LIN {X 0,Y 316.148,Z 1080.606,A -85,B 0,C 180,E1 25715.482,E2 25715.482} C_VEL
LIN {X 0,Y 359.613,Z 1022.484,A -85,B 0,C 180,E1 25721.601,E2 25721.601} C_VEL
LIN {X 0,Y 369.692,Z 1005.378,A -85,B 0,C 180,E1 25723.065,E2 25723.065} C_VEL
LIN {X 0,Y 370.148,Z 988.443,A -85,B 0,C 180,E1 25731.773,E2 25731.773} C_VEL
LIN {X 0,Y 370.715,Z 983.832,A -85,B 0,C 180,E1 25738.851,E2 25738.851} C_VEL
LIN {X 0,Y 369.808,Z 994.61,A -85,B 0,C 180,E1 25748.283,E2 25748.283} C_VEL
LIN {X 0,Y 368.373,Z 1009.498,A -85,B 0,C 180,E1 25754.057,E2 25754.057} C_VEL
LIN {X 0,Y 326.146,Z 1071.026,A -85,B 0,C 180,E1 25759.675,E2 25759.675} C_VEL
LIN {X 0,Y 280.052,Z 1123.121,A -85,B 0,C 180,E1 25768.626,E2 25768.626} C_VEL
LIN {X 0,Y 237.395,Z 1163.97,A -85,B 0,C 180,E1 25782.718,E2 25782.718} C_VEL
LIN {X 0,Y 210.63,Z 1190.183,A -85,B 0,C 180,E1 25802.091,E2 25802.091} C_VEL
LIN {X 0,Y 203.395,Z 1200.362,A -85,B 0,C 180,E1 25819.253,E2 25819.253} C_VEL
LIN {X 0,Y 203.105,Z 1202.001,A -85,B 0,C 180,E1 25832.135,E2 25832.135} C_VEL
LIN {X 0,Y 205.625,Z 1196.351,A -85,B 0,C 180,E1 25849.379,E2 25849.379} C_VEL
LIN {X 0,Y 224.205,Z 1176.349,A -85,B 0,C 180,E1 25869.979,E2 25869.979} C_VEL
LIN {X 0,Y 261.978,Z 1141.015,A -85,B 0,C 180,E1 25886.466,E2 25886.466} C_VEL
LIN {X 0,Y 308.24,Z 1092.884,A -85,B 0,C 180,E1 25897.284,E2 25897.284} C_VEL
LIN {X 0,Y 353.537,Z 1033.592,A -85,B 0,C 180,E1 25904.178,E2 25904.178} C_VEL
LIN {X 0,Y 369.486,Z 1007.292,A -85,B 0,C 180,E1 25906.321,E2 25906.321} C_VEL
LIN {X 0,Y 370.03,Z 990.826,A -85,B 0,C 180,E1 25914.09,E2 25914.09} C_VEL
LIN {X 0,Y 371.036,Z 983.808,A -85,B 0,C 180,E1 25921.148,E2 25921.148} C_VEL
LIN {X 0,Y 370.096,Z 993.398,A -85,B 0,C 180,E1 25931.209,E2 25931.209} C_VEL
LIN {X 0,Y 368.996,Z 1007.618,A -85,B 0,C 180,E1 25937.205,E2 25937.205} C_VEL
LIN {X 0,Y 326.774,Z 1068.114,A -85,B 0,C 180,E1 25942.732,E2 25942.732} C_VEL
LIN {X 0,Y 293.393,Z 1105.685,A -85,B 0,C 180,E1 25948.682,E2 25948.682} C_VEL
LIN {X 0,Y 268.809,Z 1125.767,A -85,B 0,C 180,E1 25951.921,E2 25951.921} C_VEL
LIN {X 0,Y 226.225,Z 1161.867,A -85,B 0,C 180,E1 25966.765,E2 25966.765} C_VEL
LIN {X 0,Y 202.01,Z 1181.995,A -85,B 0,C 180,E1 25985.618,E2 25985.618} C_VEL
LIN {X 0,Y 195.444,Z 1189.255,A -85,B 0,C 180,E1 26003.321,E2 26003.321} C_VEL
LIN {X 0,Y 195.404,Z 1189.222,A -85,B 0,C 180,E1 26016.69,E2 26016.69} C_VEL
LIN {X 0,Y 204.145,Z 1180,A -85,B 0,C 180,E1 26037.107,E2 26037.107} C_VEL
LIN {X 0,Y 234.232,Z 1155.422,A -85,B 0,C 180,E1 26056.755,E2 26056.755} C_VEL
LIN {X 0,Y 277.988,Z 1117.112,A -85,B 0,C 180,E1 26070.177,E2 26070.177} C_VEL
LIN {X 0,Y 325.42,Z 1066.08,A -85,B 0,C 180,E1 26078.761,E2 26078.761} C_VEL
LIN {X 0,Y 364.954,Z 1010.019,A -85,B 0,C 180,E1 26083.947,E2 26083.947} C_VEL
LIN {X 0,Y 365.855,Z 995.479,A -85,B 0,C 180,E1 26091.676,E2 26091.676} C_VEL
LIN {X 0,Y 366.492,Z 990.687,A -85,B 0,C 180,E1 26098.838,E2 26098.838} C_VEL
LIN {X 0,Y 365.305,Z 1001.773,A -85,B 0,C 180,E1 26108.386,E2 26108.386} C_VEL
LIN {X 0,Y 363.604,Z 1013.922,A -85,B 0,C 180,E1 26113.125,E2 26113.125} C_VEL
LIN {X 0,Y 318.765,Z 1076.531,A -85,B 0,C 180,E1 26118.987,E2 26118.987} C_VEL
LIN {X 0,Y 271.684,Z 1127.247,A -85,B 0,C 180,E1 26128.161,E2 26128.161} C_VEL
LIN {X 0,Y 227.974,Z 1166.993,A -85,B 0,C 180,E1 26142.962,E2 26142.962} C_VEL
LIN {X 0,Y 201.693,Z 1191.616,A -85,B 0,C 180,E1 26163.179,E2 26163.179} C_VEL
LIN {X 0,Y 195.081,Z 1201.22,A -85,B 0,C 180,E1 26183.299,E2 26183.299} C_VEL
LIN {X 0,Y 195.077,Z 1201.233,A -85,B 0,C 180,E1 26196.692,E2 26196.692} C_VEL
LIN {X 0,Y 200.185,Z 1193.301,A -85,B 0,C 180,E1 26214.619,E2 26214.619} C_VEL
LIN {X 0,Y 224.297,Z 1170.256,A -85,B 0,C 180,E1 26235.223,E2 26235.223} C_VEL
LIN {X 0,Y 265.902,Z 1132.749,A -85,B 0,C 180,E1 26250.423,E2 26250.423} C_VEL
LIN {X 0,Y 314.147,Z 1082.127,A -85,B 0,C 180,E1 26260.27,E2 26260.27} C_VEL
LIN {X 0,Y 359.015,Z 1021.48,A -85,B 0,C 180,E1 26266.376,E2 26266.376} C_VEL
LIN {X 0,Y 364.771,Z 1011.464,A -85,B 0,C 180,E1 26267.357,E2 26267.357} C_VEL
LIN {X 0,Y 365.816,Z 996.158,A -85,B 0,C 180,E1 26275.216,E2 26275.216} C_VEL
LIN {X 0,Y 366.821,Z 990.653,A -85,B 0,C 180,E1 26281.161,E2 26281.161} C_VEL
LIN {X 0,Y 365.711,Z 999.528,A -85,B 0,C 180,E1 26290.739,E2 26290.739} C_VEL
LIN {X 0,Y 364.587,Z 1011.509,A -85,B 0,C 180,E1 26296.224,E2 26296.224} C_VEL
LIN {X 0,Y 320.68,Z 1072.197,A -85,B 0,C 180,E1 26301.87,E2 26301.87} C_VEL
LIN {X 0,Y 273.521,Z 1121.485,A -85,B 0,C 180,E1 26310.759,E2 26310.759} C_VEL
LIN {X 0,Y 268.809,Z 1125.767,A -85,B 0,C 180,E1 26311.921,E2 26311.921} C_VEL
LIN {X 0,Y 244.101,Z 1143.39,A -85,B 0,C 180,E1 26316.075,E2 26316.075} C_VEL
LIN {X 0,Y 205.94,Z 1173.133,A -85,B 0,C 180,E1 26333.787,E2 26333.787} C_VEL
LIN {X 0,Y 189.446,Z 1186.942,A -85,B 0,C 180,E1 26353.734,E2 26353.734} C_VEL
LIN {X 0,Y 187.43,Z 1189.94,A -85,B 0,C 180,E1 26372.323,E2 26372.323} C_VEL
LIN {X 0,Y 192.941,Z 1183.622,A -85,B 0,C 180,E1 26393.146,E2 26393.146} C_VEL
LIN {X 0,Y 218.988,Z 1163.089,A -85,B 0,C 180,E1 26413.976,E2 26413.976} C_VEL
LIN {X 0,Y 262.449,Z 1127.725,A -85,B 0,C 180,E1 26429.025,E2 26429.025} C_VEL
LIN {X 0,Y 311.303,Z 1079.422,A -85,B 0,C 180,E1 26438.481,E2 26438.481} C_VEL
LIN {X 0,Y 356.624,Z 1020.527,A -85,B 0,C 180,E1 26444.269,E2 26444.269} C_VEL
LIN {X 0,Y 360.249,Z 1014.774,A -85,B 0,C 180,E1 26444.806,E2 26444.806} C_VEL
LIN {X 0,Y 361.457,Z 1001.135,A -85,B 0,C 180,E1 26452.788,E2 26452.788} C_VEL
LIN {X 0,Y 362.265,Z 997.544,A -85,B 0,C 180,E1 26458.824,E2 26458.824} C_VEL
LIN {X 0,Y 360.713,Z 1007.612,A -85,B 0,C 180,E1 26467.885,E2 26467.885} C_VEL
LIN {X 0,Y 358.795,Z 1018.34,A -85,B 0,C 180,E1 26472.177,E2 26472.177} C_VEL
LIN {X 0,Y 312.986,Z 1079.796,A -85,B 0,C 180,E1 26478.022,E2 26478.022} C_VEL
LIN {X 0,Y 264.611,Z 1129.862,A -85,B 0,C 180,E1 26487.33,E2 26487.33} C_VEL
LIN {X 0,Y 220.325,Z 1168.374,A -85,B 0,C 180,E1 26502.322,E2 26502.322} C_VEL
LIN {X 0,Y 194.323,Z 1191.359,A -85,B 0,C 180,E1 26522.075,E2 26522.075} C_VEL
LIN {X 0,Y 187.07,Z 1200.971,A -85,B 0,C 180,E1 26543.011,E2 26543.011} C_VEL
LIN {X 0,Y 187.066,Z 1200.984,A -85,B 0,C 180,E1 26556.98,E2 26556.98} C_VEL
LIN {X 0,Y 192.676,Z 1193.044,A -85,B 0,C 180,E1 26575.646,E2 26575.646} C_VEL
LIN {X 0,Y 218.416,Z 1169.988,A -85,B 0,C 180,E1 26596.8,E2 26596.8} C_VEL
LIN {X 0,Y 261.83,Z 1132.468,A -85,B 0,C 180,E1 26612.033,E2 26612.033} C_VEL
LIN {X 0,Y 311.426,Z 1081.82,A -85,B 0,C 180,E1 26621.717,E2 26621.717} C_VEL
LIN {X 0,Y 357.409,Z 1020.732,A -85,B 0,C 180,E1 26627.691,E2 26627.691} C_VEL
LIN {X 0,Y 360.11,Z 1015.85,A -85,B 0,C 180,E1 26628.363,E2 26628.363} C_VEL
LIN {X 0,Y 361.546,Z 1001.58,A -85,B 0,C 180,E1 26636.365,E2 26636.365} C_VEL
LIN {X 0,Y 362.6,Z 997.505,A -85,B 0,C 180,E1 26641.175,E2 26641.175} C_VEL
LIN {X 0,Y 361.062,Z 1006.48,A -85,B 0,C 180,E1 26650.879,E2 26650.879} C_VEL
LIN {X 0,Y 359.569,Z 1016.385,A -85,B 0,C 180,E1 26655.305,E2 26655.305} C_VEL
LIN {X 0,Y 314.729,Z 1075.84,A -85,B 0,C 180,E1 26660.939,E2 26660.939} C_VEL
LIN {X 0,Y 266.707,Z 1124.112,A -85,B 0,C 180,E1 26669.88,E2 26669.88} C_VEL
LIN {X 0,Y 244.101,Z 1143.39,A -85,B 0,C 180,E1 26676.075,E2 26676.075} C_VEL
LIN {X 0,Y 219.813,Z 1158.391,A -85,B 0,C 180,E1 26681.306,E2 26681.306} C_VEL
LIN {X 0,Y 188.769,Z 1181.284,A -85,B 0,C 180,E1 26701.682,E2 26701.682} C_VEL
LIN {X 0,Y 179.487,Z 1189.751,A -85,B 0,C 180,E1 26722.724,E2 26722.724} C_VEL
LIN {X 0,Y 179.428,Z 1189.721,A -85,B 0,C 180,E1 26737.288,E2 26737.288} C_VEL
LIN {X 0,Y 188.648,Z 1181.254,A -85,B 0,C 180,E1 26758.235,E2 26758.235} C_VEL
LIN {X 0,Y 219.961,Z 1158.336,A -85,B 0,C 180,E1 26778.52,E2 26778.52} C_VEL
LIN {X 0,Y 265.657,Z 1121.739,A -85,B 0,C 180,E1 26792.237,E2 26792.237} C_VEL
LIN {X 0,Y 315.107,Z 1072.386,A -85,B 0,C 180,E1 26800.828,E2 26800.828} C_VEL
LIN {X 0,Y 355.471,Z 1019.161,A -85,B 0,C 180,E1 26805.802,E2 26805.802} C_VEL
LIN {X 0,Y 356.974,Z 1006.833,A -85,B 0,C 180,E1 26813.923,E2 26813.923} C_VEL
LIN {X 0,Y 357.809,Z 1004.236,A -85,B 0,C 180,E1 26818.81,E2 26818.81} C_VEL
LIN {X 0,Y 355.979,Z 1014.642,A -85,B 0,C 180,E1 26827.99,E2 26827.99} C_VEL
LIN {X 0,Y 353.349,Z 1023.665,A -85,B 0,C 180,E1 26831.284,E2 26831.284} C_VEL
LIN {X 0,Y 306.092,Z 1084.408,A -85,B 0,C 180,E1 26837.196,E2 26837.196} C_VEL
LIN {X 0,Y 255.588,Z 1134.273,A -85,B 0,C 180,E1 26846.934,E2 26846.934} C_VEL
LIN {X 0,Y 210.554,Z 1171.596,A -85,B 0,C 180,E1 26862.763,E2 26862.763} C_VEL
LIN {X 0,Y 184.361,Z 1193.782,A -85,B 0,C 180,E1 26884.749,E2 26884.749} C_VEL
LIN {X 0,Y 179.061,Z 1200.721,A -85,B 0,C 180,E1 26902.697,E2 26902.697} C_VEL
LIN {X 0,Y 179.057,Z 1200.734,A -85,B 0,C 180,E1 26917.294,E2 26917.294} C_VEL
LIN {X 0,Y 185.211,Z 1192.786,A -85,B 0,C 180,E1 26936.76,E2 26936.76} C_VEL
LIN {X 0,Y 211.478,Z 1170.765,A -85,B 0,C 180,E1 26957.828,E2 26957.828} C_VEL
LIN {X 0,Y 256.495,Z 1133.534,A -85,B 0,C 180,E1 26973.322,E2 26973.322} C_VEL
LIN {X 0,Y 307.722,Z 1082.846,A -85,B 0,C 180,E1 26983.012,E2 26983.012} C_VEL
LIN {X 0,Y 354.488,Z 1022.232,A -85,B 0,C 180,E1 26988.865,E2 26988.865} C_VEL
LIN {X 0,Y 356.76,Z 1009.616,A -85,B 0,C 180,E1 26995.293,E2 26995.293} C_VEL
LIN {X 0,Y 358.136,Z 1004.212,A -85,B 0,C 180,E1 27001.189,E2 27001.189} C_VEL
LIN {X 0,Y 356.382,Z 1013.484,A -85,B 0,C 180,E1 27011.024,E2 27011.024} C_VEL
LIN {X 0,Y 354.227,Z 1021.652,A -85,B 0,C 180,E1 27014.403,E2 27014.403} C_VEL
LIN {X 0,Y 307.535,Z 1080.944,A -85,B 0,C 180,E1 27020.17,E2 27020.17} C_VEL
LIN {X 0,Y 258.599,Z 1127.919,A -85,B 0,C 180,E1 27029.278,E2 27029.278} C_VEL
LIN {X 0,Y 219.813,Z 1158.391,A -85,B 0,C 180,E1 27041.306,E2 27041.306} C_VEL
LIN {X 0,Y 197.353,Z 1170.633,A -85,B 0,C 180,E1 27048.102,E2 27048.102} C_VEL
LIN {X 0,Y 175.069,Z 1186.508,A -85,B 0,C 180,E1 27069.732,E2 27069.732} C_VEL
LIN {X 0,Y 171.299,Z 1190.45,A -85,B 0,C 180,E1 27087.468,E2 27087.468} C_VEL
LIN {X 0,Y 174.006,Z 1187.386,A -85,B 0,C 180,E1 27107.766,E2 27107.766} C_VEL
LIN {X 0,Y 195.922,Z 1171.396,A -85,B 0,C 180,E1 27131.148,E2 27131.148} C_VEL
LIN {X 0,Y 237.45,Z 1141.724,A -85,B 0,C 180,E1 27147.944,E2 27147.944} C_VEL
LIN {X 0,Y 288.79,Z 1097.502,A -85,B 0,C 180,E1 27158.773,E2 27158.773} C_VEL
LIN {X 0,Y 338.132,Z 1041.454,A -85,B 0,C 180,E1 27165.325,E2 27165.325} C_VEL
LIN {X 0,Y 350.672,Z 1023.964,A -85,B 0,C 180,E1 27166.674,E2 27166.674} C_VEL
LIN {X 0,Y 352.423,Z 1013.558,A -85,B 0,C 180,E1 27173.844,E2 27173.844} C_VEL
LIN {X 0,Y 353.285,Z 1010.885,A -85,B 0,C 180,E1 27178.794,E2 27178.794} C_VEL
LIN {X 0,Y 350.984,Z 1021.49,A -85,B 0,C 180,E1 27188.105,E2 27188.105} C_VEL
LIN {X 0,Y 348.689,Z 1027.918,A -85,B 0,C 180,E1 27190.271,E2 27190.271} C_VEL
LIN {X 0,Y 300.52,Z 1087.644,A -85,B 0,C 180,E1 27196.159,E2 27196.159} C_VEL
LIN {X 0,Y 248.199,Z 1137.19,A -85,B 0,C 180,E1 27206.136,E2 27206.136} C_VEL
LIN {X 0,Y 203.005,Z 1172.745,A -85,B 0,C 180,E1 27222.015,E2 27222.015} C_VEL
LIN {X 0,Y 176.089,Z 1194.236,A -85,B 0,C 180,E1 27244.949,E2 27244.949} C_VEL
LIN {X 0,Y 171.066,Z 1200.471,A -85,B 0,C 180,E1 27262.353,E2 27262.353} C_VEL
LIN {X 0,Y 171.062,Z 1200.485,A -85,B 0,C 180,E1 27277.637,E2 27277.637} C_VEL
LIN {X 0,Y 177.851,Z 1192.53,A -85,B 0,C 180,E1 27297.962,E2 27297.962} C_VEL
LIN {X 0,Y 207.26,Z 1169.459,A -85,B 0,C 180,E1 27320.193,E2 27320.193} C_VEL
LIN {X 0,Y 255.166,Z 1131.238,A -85,B 0,C 180,E1 27335.556,E2 27335.556} C_VEL
LIN {X 0,Y 306.592,Z 1081.211,A -85,B 0,C 180,E1 27344.685,E2 27344.685} C_VEL
LIN {X 0,Y 350.515,Z 1025.296,A -85,B 0,C 180,E1 27350.067,E2 27350.067} C_VEL
LIN {X 0,Y 352.797,Z 1012.784,A -85,B 0,C 180,E1 27358.742,E2 27358.742} C_VEL
LIN {X 0,Y 352.914,Z 1012.124,A -85,B 0,C 180,E1 27363.674,E2 27363.674} C_VEL
LIN {X 0,Y 350.965,Z 1022.787,A -85,B 0,C 180,E1 27372.502,E2 27372.502} C_VEL
LIN {X 0,Y 349.511,Z 1026.126,A -85,B 0,C 180,E1 27373.417,E2 27373.417} C_VEL
LIN {X 0,Y 301.887,Z 1084.419,A -85,B 0,C 180,E1 27379.146,E2 27379.146} C_VEL
LIN {X 0,Y 250.529,Z 1131.65,A -85,B 0,C 180,E1 27388.639,E2 27388.639} C_VEL
LIN {X 0,Y 205.093,Z 1165.26,A -85,B 0,C 180,E1 27403.874,E2 27403.874} C_VEL
LIN {X 0,Y 197.353,Z 1170.633,A -85,B 0,C 180,E1 27408.102,E2 27408.102} C_VEL
LIN {X 0,Y 177.075,Z 1180.099,A -85,B 0,C 180,E1 27416.564,E2 27416.564} C_VEL
LIN {X 0,Y 164.44,Z 1189.285,A -85,B 0,C 180,E1 27436.676,E2 27436.676} C_VEL
LIN {X 0,Y 163.401,Z 1190.683,A -85,B 0,C 180,E1 27452.665,E2 27452.665} C_VEL
LIN {X 0,Y 170.599,Z 1184.429,A -85,B 0,C 180,E1 27476.273,E2 27476.273} C_VEL
LIN {X 0,Y 201.697,Z 1164.027,A -85,B 0,C 180,E1 27498.76,E2 27498.76} C_VEL
LIN {X 0,Y 249.635,Z 1129.369,A -85,B 0,C 180,E1 27513.651,E2 27513.651} C_VEL
LIN {X 0,Y 301.498,Z 1082.119,A -85,B 0,C 180,E1 27522.562,E2 27522.562} C_VEL
LIN {X 0,Y 346.074,Z 1027.998,A -85,B 0,C 180,E1 27527.996,E2 27527.996} C_VEL
LIN {X 0,Y 348.156,Z 1018.32,A -85,B 0,C 180,E1 27536.276,E2 27536.276} C_VEL
LIN {X 0,Y 347.866,Z 1019.205,A -85,B 0,C 180,E1 27541.276,E2 27541.276} C_VEL
LIN {X 0,Y 345.552,Z 1030.072,A -85,B 0,C 180,E1 27549.071,E2 27549.071} C_VEL
LIN {X 0,Y 295.713,Z 1090.045,A -85,B 0,C 180,E1 27554.976,E2 27554.976} C_VEL
LIN {X 0,Y 242.416,Z 1138.628,A -85,B 0,C 180,E1 27564.885,E2 27564.885} C_VEL
LIN {X 0,Y 194.887,Z 1174.275,A -85,B 0,C 180,E1 27581.513,E2 27581.513} C_VEL
LIN {X 0,Y 167.396,Z 1195.046,A -85,B 0,C 180,E1 27605.935,E2 27605.935} C_VEL
LIN {X 0,Y 163.212,Z 1200.763,A -85,B 0,C 180,E1 27627.332,E2 27627.332} C_VEL
LIN {X 0,Y 163.694,Z 1199.123,A -85,B 0,C 180,E1 27643.386,E2 27643.386} C_VEL
LIN {X 0,Y 178.726,Z 1185.905,A -85,B 0,C 180,E1 27667.958,E2 27667.958} C_VEL
LIN {X 0,Y 217.781,Z 1157.795,A -85,B 0,C 180,E1 27688.054,E2 27688.054} C_VEL
LIN {X 0,Y 269.121,Z 1115.976,A -85,B 0,C 180,E1 27700.702,E2 27700.702} C_VEL
LIN {X 0,Y 321.265,Z 1061.956,A -85,B 0,C 180,E1 27708.285,E2 27708.285} C_VEL
LIN {X 0,Y 345.857,Z 1029.699,A -85,B 0,C 180,E1 27711.138,E2 27711.138} C_VEL
LIN {X 0,Y 348.062,Z 1019.342,A -85,B 0,C 180,E1 27718.725,E2 27718.725} C_VEL
LIN {X 0,Y 348.201,Z 1018.692,A -85,B 0,C 180,E1 27723.723,E2 27723.723} C_VEL
LIN {X 0,Y 345.992,Z 1028.957,A -85,B 0,C 180,E1 27732.259,E2 27732.259} C_VEL
LIN {X 0,Y 296.664,Z 1087.399,A -85,B 0,C 180,E1 27738.035,E2 27738.035} C_VEL
LIN {X 0,Y 245.226,Z 1133.012,A -85,B 0,C 180,E1 27747.293,E2 27747.293} C_VEL
LIN {X 0,Y 197.439,Z 1166.813,A -85,B 0,C 180,E1 27763.146,E2 27763.146} C_VEL
LIN {X 0,Y 177.075,Z 1180.099,A -85,B 0,C 180,E1 27776.564,E2 27776.564} C_VEL
LIN {X 0,Y 160.31,Z 1186.702,A -85,B 0,C 180,E1 27786.989,E2 27786.989} C_VEL
LIN {X 0,Y 155.28,Z 1190.945,A -85,B 0,C 180,E1 27807.207,E2 27807.207} C_VEL
LIN {X 0,Y 158.613,Z 1187.888,A -85,B 0,C 180,E1 27829.556,E2 27829.556} C_VEL
LIN {X 0,Y 183.833,Z 1171.909,A -85,B 0,C 180,E1 27854.53,E2 27854.53} C_VEL
LIN {X 0,Y 228.902,Z 1142.399,A -85,B 0,C 180,E1 27871.39,E2 27871.39} C_VEL
LIN {X 0,Y 283.283,Z 1098.089,A -85,B 0,C 180,E1 27881.855,E2 27881.855} C_VEL
LIN {X 0,Y 334.214,Z 1042.379,A -85,B 0,C 180,E1 27887.997,E2 27887.997} C_VEL
LIN {X 0,Y 341.349,Z 1032.559,A -85,B 0,C 180,E1 27889.062,E2 27889.062} C_VEL
LIN {X 0,Y 343.423,Z 1024.484,A -85,B 0,C 180,E1 27897.097,E2 27897.097} C_VEL
LIN {X 0,Y 342.232,Z 1028.788,A -85,B 0,C 180,E1 27904.384,E2 27904.384} C_VEL
LIN {X 0,Y 340.123,Z 1035.463,A -85,B 0,C 180,E1 27908.143,E2 27908.143} C_VEL
LIN {X 0,Y 289.167,Z 1094.136,A -85,B 0,C 180,E1 27914.007,E2 27914.007} C_VEL
LIN {X 0,Y 234.775,Z 1141.61,A -85,B 0,C 180,E1 27924.061,E2 27924.061} C_VEL
LIN {X 0,Y 186.401,Z 1176.078,A -85,B 0,C 180,E1 27941.181,E2 27941.181} C_VEL
LIN {X 0,Y 159.909,Z 1194.791,A -85,B 0,C 180,E1 27964.732,E2 27964.732} C_VEL
LIN {X 0,Y 155.193,Z 1200.515,A -85,B 0,C 180,E1 27987.194,E2 27987.194} C_VEL
LIN {X 0,Y 155.786,Z 1198.872,A -85,B 0,C 180,E1 28004.079,E2 28004.079} C_VEL
LIN {X 0,Y 172.246,Z 1185.648,A -85,B 0,C 180,E1 28029.66,E2 28029.66} C_VEL
LIN {X 0,Y 215.14,Z 1156.359,A -85,B 0,C 180,E1 28050.512,E2 28050.512} C_VEL
LIN {X 0,Y 268.052,Z 1114.339,A -85,B 0,C 180,E1 28062.679,E2 28062.679} C_VEL
LIN {X 0,Y 320.643,Z 1060.484,A -85,B 0,C 180,E1 28069.851,E2 28069.851} C_VEL
LIN {X 0,Y 341.192,Z 1034.02,A -85,B 0,C 180,E1 28072.244,E2 28072.244} C_VEL
LIN {X 0,Y 344.158,Z 1023.885,A -85,B 0,C 180,E1 28081.238,E2 28081.238} C_VEL
LIN {X 0,Y 341.599,Z 1032.097,A -85,B 0,C 180,E1 28090.399,E2 28090.399} C_VEL
LIN {X 0,Y 338.689,Z 1036.85,A -85,B 0,C 180,E1 28091.51,E2 28091.51} C_VEL
LIN {X 0,Y 287.992,Z 1093.71,A -85,B 0,C 180,E1 28097.374,E2 28097.374} C_VEL
LIN {X 0,Y 234.647,Z 1138.428,A -85,B 0,C 180,E1 28107.175,E2 28107.175} C_VEL
LIN {X 0,Y 188.083,Z 1169.48,A -85,B 0,C 180,E1 28123.244,E2 28123.244} C_VEL
LIN {X 0,Y 160.31,Z 1186.702,A -85,B 0,C 180,E1 28146.989,E2 28146.989} C_VEL
LIN {X 0,Y 147.799,Z 1190.449,A -85,B 0,C 180,E1 28159.315,E2 28159.315} C_VEL
LIN {X 0,Y 147.555,Z 1190.716,A -85,B 0,C 180,E1 28178.874,E2 28178.874} C_VEL
LIN {X 0,Y 161.187,Z 1181.92,A -85,B 0,C 180,E1 28204.374,E2 28204.374} C_VEL
LIN {X 0,Y 201.291,Z 1158.378,A -85,B 0,C 180,E1 28226.229,E2 28226.229} C_VEL
LIN {X 0,Y 253.585,Z 1121.644,A -85,B 0,C 180,E1 28239.144,E2 28239.144} C_VEL
LIN {X 0,Y 307.659,Z 1071.746,A -85,B 0,C 180,E1 28246.807,E2 28246.807} C_VEL
LIN {X 0,Y 336.43,Z 1037.605,A -85,B 0,C 180,E1 28249.881,E2 28249.881} C_VEL
LIN {X 0,Y 339.02,Z 1030.333,A -85,B 0,C 180,E1 28258.744,E2 28258.744} C_VEL
LIN {X 0,Y 336.112,Z 1038.748,A -85,B 0,C 180,E1 28266.849,E2 28266.849} C_VEL
LIN {X 0,Y 283.878,Z 1097.101,A -85,B 0,C 180,E1 28272.841,E2 28272.841} C_VEL
LIN {X 0,Y 228.398,Z 1143.654,A -85,B 0,C 180,E1 28282.878,E2 28282.878} C_VEL
LIN {X 0,Y 179.728,Z 1176.629,A -85,B 0,C 180,E1 28299.808,E2 28299.808} C_VEL
LIN {X 0,Y 150.937,Z 1195.819,A -85,B 0,C 180,E1 28326.307,E2 28326.307} C_VEL
LIN {X 0,Y 147.162,Z 1200.267,A -85,B 0,C 180,E1 28347.041,E2 28347.041} C_VEL
LIN {X 0,Y 147.911,Z 1198.621,A -85,B 0,C 180,E1 28364.846,E2 28364.846} C_VEL
LIN {X 0,Y 165.904,Z 1185.39,A -85,B 0,C 180,E1 28391.5,E2 28391.5} C_VEL
LIN {X 0,Y 210.263,Z 1156.652,A -85,B 0,C 180,E1 28412.254,E2 28412.254} C_VEL
LIN {X 0,Y 265.007,Z 1114.613,A -85,B 0,C 180,E1 28424.301,E2 28424.301} C_VEL
LIN {X 0,Y 318.771,Z 1060.775,A -85,B 0,C 180,E1 28431.267,E2 28431.267} C_VEL
LIN {X 0,Y 336.315,Z 1038.815,A -85,B 0,C 180,E1 28433.17,E2 28433.17} C_VEL
LIN {X 0,Y 339.336,Z 1030.325,A -85,B 0,C 180,E1 28441.255,E2 28441.255} C_VEL
LIN {X 0,Y 336.497,Z 1037.893,A -85,B 0,C 180,E1 28450.066,E2 28450.066} C_VEL
LIN {X 0,Y 285.659,Z 1093.995,A -85,B 0,C 180,E1 28455.81,E2 28455.81} C_VEL
LIN {X 0,Y 231.888,Z 1138.032,A -85,B 0,C 180,E1 28465.137,E2 28465.137} C_VEL
LIN {X 0,Y 182.519,Z 1169.738,A -85,B 0,C 180,E1 28481.354,E2 28481.354} C_VEL
LIN {X 0,Y 152.408,Z 1187.262,A -85,B 0,C 180,E1 28506.552,E2 28506.552} C_VEL
LIN {X 0,Y 147.799,Z 1190.449,A -85,B 0,C 180,E1 28519.315,E2 28519.315} C_VEL
LIN {X 0,Y 139.376,Z 1191.423,A -85,B 0,C 180,E1 28533.177,E2 28533.177} C_VEL
LIN {X 0,Y 148.389,Z 1185.48,A -85,B 0,C 180,E1 28559.729,E2 28559.729} C_VEL
LIN {X 0,Y 186.354,Z 1164.807,A -85,B 0,C 180,E1 28584.475,E2 28584.475} C_VEL
LIN {X 0,Y 240.58,Z 1129.535,A -85,B 0,C 180,E1 28599.102,E2 28599.102} C_VEL
LIN {X 0,Y 295.557,Z 1082.561,A -85,B 0,C 180,E1 28607.147,E2 28607.147} C_VEL
LIN {X 0,Y 331.618,Z 1042.53,A -85,B 0,C 180,E1 28610.809,E2 28610.809} C_VEL
LIN {X 0,Y 333.925,Z 1036.578,A -85,B 0,C 180,E1 28618.724,E2 28618.724} C_VEL
LIN {X 0,Y 330.366,Z 1044.837,A -85,B 0,C 180,E1 28626.042,E2 28626.042} C_VEL
LIN {X 0,Y 277.016,Z 1101.67,A -85,B 0,C 180,E1 28631.871,E2 28631.871} C_VEL
LIN {X 0,Y 220.742,Z 1146.603,A -85,B 0,C 180,E1 28641.948,E2 28641.948} C_VEL
LIN {X 0,Y 172.467,Z 1177.612,A -85,B 0,C 180,E1 28658.703,E2 28658.703} C_VEL
LIN {X 0,Y 144.202,Z 1194.981,A -85,B 0,C 180,E1 28683.605,E2 28683.605} C_VEL
LIN {X 0,Y 139.153,Z 1200.019,A -85,B 0,C 180,E1 28706.87,E2 28706.87} C_VEL
LIN {X 0,Y 140.045,Z 1198.37,A -85,B 0,C 180,E1 28725.701,E2 28725.701} C_VEL
LIN {X 0,Y 159.745,Z 1185.132,A -85,B 0,C 180,E1 28753.485,E2 28753.485} C_VEL
LIN {X 0,Y 206.79,Z 1156.157,A -85,B 0,C 180,E1 28774.449,E2 28774.449} C_VEL
LIN {X 0,Y 263.773,Z 1113.575,A -85,B 0,C 180,E1 28786.213,E2 28786.213} C_VEL
LIN {X 0,Y 319.344,Z 1058.362,A -85,B 0,C 180,E1 28792.938,E2 28792.938} C_VEL
LIN {X 0,Y 331.584,Z 1043.291,A -85,B 0,C 180,E1 28794.387,E2 28794.387} C_VEL
LIN {X 0,Y 334.24,Z 1036.57,A -85,B 0,C 180,E1 28801.274,E2 28801.274} C_VEL
LIN {X 0,Y 331.179,Z 1043.489,A -85,B 0,C 180,E1 28809.203,E2 28809.203} C_VEL
LIN {X 0,Y 278.259,Z 1099.2,A -85,B 0,C 180,E1 28814.906,E2 28814.906} C_VEL
LIN {X 0,Y 221.469,Z 1143.13,A -85,B 0,C 180,E1 28824.875,E2 28824.875} C_VEL
LIN {X 0,Y 170.456,Z 1173.66,A -85,B 0,C 180,E1 28842.786,E2 28842.786} C_VEL
LIN {X 0,Y 143.331,Z 1188.443,A -85,B 0,C 180,E1 28868.271,E2 28868.271} C_VEL
LIN {X 0,Y 139.376,Z 1191.423,A -85,B 0,C 180,E1 28893.177,E2 28893.177} C_VEL
LIN {X 0,Y 133.609,Z 1189.902,A -85,B 0,C 180,E1 28907.967,E2 28907.967} C_VEL
LIN {X 0,Y 160.63,Z 1176.013,A -85,B 0,C 180,E1 28937.035,E2 28937.035} C_VEL
LIN {X 0,Y 212.109,Z 1147.013,A -85,B 0,C 180,E1 28955.735,E2 28955.735} C_VEL
LIN {X 0,Y 270.507,Z 1104.137,A -85,B 0,C 180,E1 28965.924,E2 28965.924} C_VEL
LIN {X 0,Y 324.203,Z 1050.319,A -85,B 0,C 180,E1 28971.645,E2 28971.645} C_VEL
LIN {X 0,Y 326.87,Z 1047.026,A -85,B 0,C 180,E1 28972.168,E2 28972.168} C_VEL
LIN {X 0,Y 328.821,Z 1042.79,A -85,B 0,C 180,E1 28978.705,E2 28978.705} C_VEL
LIN {X 0,Y 325.732,Z 1049.163,A -85,B 0,C 180,E1 28984.94,E2 28984.94} C_VEL
LIN {X 0,Y 271.805,Z 1104.478,A -85,B 0,C 180,E1 28990.624,E2 28990.624} C_VEL
LIN {X 0,Y 214.328,Z 1148.539,A -85,B 0,C 180,E1 29000.643,E2 29000.643} C_VEL
LIN {X 0,Y 161.767,Z 1180.334,A -85,B 0,C 180,E1 29019.33,E2 29019.33} C_VEL
LIN {X 0,Y 134.492,Z 1196.323,A -85,B 0,C 180,E1 29046.749,E2 29046.749} C_VEL
LIN {X 0,Y 131.119,Z 1199.77,A -85,B 0,C 180,E1 29066.678,E2 29066.678} C_VEL
LIN {X 0,Y 132.216,Z 1198.119,A -85,B 0,C 180,E1 29086.657,E2 29086.657} C_VEL
LIN {X 0,Y 153.787,Z 1184.874,A -85,B 0,C 180,E1 29115.629,E2 29115.629} C_VEL
LIN {X 0,Y 203.326,Z 1155.855,A -85,B 0,C 180,E1 29136.628,E2 29136.628} C_VEL
LIN {X 0,Y 262.039,Z 1113.167,A -85,B 0,C 180,E1 29148.027,E2 29148.027} C_VEL
LIN {X 0,Y 318.095,Z 1058.429,A -85,B 0,C 180,E1 29154.387,E2 29154.387} C_VEL
LIN {X 0,Y 326.732,Z 1048.058,A -85,B 0,C 180,E1 29155.476,E2 29155.476} C_VEL
LIN {X 0,Y 329.121,Z 1042.799,A -85,B 0,C 180,E1 29161.294,E2 29161.294} C_VEL
LIN {X 0,Y 325.59,Z 1049.035,A -85,B 0,C 180,E1 29168.172,E2 29168.172} C_VEL
LIN {X 0,Y 271.625,Z 1103.397,A -85,B 0,C 180,E1 29173.85,E2 29173.85} C_VEL
LIN {X 0,Y 215.113,Z 1145.301,A -85,B 0,C 180,E1 29183.593,E2 29183.593} C_VEL
LIN {X 0,Y 162.82,Z 1175.026,A -85,B 0,C 180,E1 29201.838,E2 29201.838} C_VEL
LIN {X 0,Y 135.806,Z 1188.694,A -85,B 0,C 180,E1 29227,E2 29227} C_VEL
LIN {X 0,Y 131.364,Z 1191.675,A -85,B 0,C 180,E1 29253.316,E2 29253.316} C_VEL
LIN {X 0,Y 133.609,Z 1189.902,A -85,B 0,C 180,E1 29267.967,E2 29267.967} C_VEL
LIN {X 0,Y 134.399,Z 1186.002,A -85,B 0,C 180,E1 29283.137,E2 29283.137} C_VEL
LIN {X 0,Y 176.036,Z 1165.948,A -85,B 0,C 180,E1 29308.37,E2 29308.37} C_VEL
LIN {X 0,Y 232.953,Z 1131.721,A -85,B 0,C 180,E1 29322.463,E2 29322.463} C_VEL
LIN {X 0,Y 290.598,Z 1084.896,A -85,B 0,C 180,E1 29330.084,E2 29330.084} C_VEL
LIN {X 0,Y 321.865,Z 1051.94,A -85,B 0,C 180,E1 29333.257,E2 29333.257} C_VEL
LIN {X 0,Y 323.566,Z 1048.895,A -85,B 0,C 180,E1 29338.684,E2 29338.684} C_VEL
LIN {X 0,Y 320.855,Z 1053.77,A -85,B 0,C 180,E1 29343.834,E2 29343.834} C_VEL
LIN {X 0,Y 265.07,Z 1108.686,A -85,B 0,C 180,E1 29349.528,E2 29349.528} C_VEL
LIN {X 0,Y 205.454,Z 1152.139,A -85,B 0,C 180,E1 29359.855,E2 29359.855} C_VEL
LIN {X 0,Y 152.111,Z 1182.46,A -85,B 0,C 180,E1 29379.398,E2 29379.398} C_VEL
LIN {X 0,Y 126.977,Z 1196.069,A -85,B 0,C 180,E1 29405.283,E2 29405.283} C_VEL
LIN {X 0,Y 123.093,Z 1199.522,A -85,B 0,C 180,E1 29426.461,E2 29426.461} C_VEL
LIN {X 0,Y 124.417,Z 1197.867,A -85,B 0,C 180,E1 29447.734,E2 29447.734} C_VEL
LIN {X 0,Y 148.733,Z 1184.288,A -85,B 0,C 180,E1 29478.366,E2 29478.366} C_VEL
LIN {X 0,Y 200.281,Z 1155.473,A -85,B 0,C 180,E1 29498.923,E2 29498.923} C_VEL
LIN {X 0,Y 260.147,Z 1113.109,A -85,B 0,C 180,E1 29509.802,E2 29509.802} C_VEL
LIN {X 0,Y 317.018,Z 1058.529,A -85,B 0,C 180,E1 29515.854,E2 29515.854} C_VEL
LIN {X 0,Y 321.777,Z 1052.802,A -85,B 0,C 180,E1 29516.592,E2 29516.592} C_VEL
LIN {X 0,Y 323.859,Z 1048.91,A -85,B 0,C 180,E1 29521.315,E2 29521.315} C_VEL
LIN {X 0,Y 320.534,Z 1053.952,A -85,B 0,C 180,E1 29527.073,E2 29527.073} C_VEL
LIN {X 0,Y 264.393,Z 1108.181,A -85,B 0,C 180,E1 29532.83,E2 29532.83} C_VEL
LIN {X 0,Y 205.82,Z 1149.382,A -85,B 0,C 180,E1 29542.935,E2 29542.935} C_VEL
LIN {X 0,Y 153.058,Z 1177.441,A -85,B 0,C 180,E1 29562.012,E2 29562.012} C_VEL
LIN {X 0,Y 125.403,Z 1190.532,A -85,B 0,C 180,E1 29592.41,E2 29592.41} C_VEL
LIN {X 0,Y 123.346,Z 1191.923,A -85,B 0,C 180,E1 29613.531,E2 29613.531} C_VEL
LIN {X 0,Y 134.399,Z 1186.002,A -85,B 0,C 180,E1 29643.137,E2 29643.137} C_VEL
LIN {X 0,Y 142.409,Z 1179.823,A -85,B 0,C 180,E1 29657.294,E2 29657.294} C_VEL
LIN {X 0,Y 196.285,Z 1153.115,A -85,B 0,C 180,E1 29677.765,E2 29677.765} C_VEL
LIN {X 0,Y 257.383,Z 1112.482,A -85,B 0,C 180,E1 29688.198,E2 29688.198} C_VEL
LIN {X 0,Y 314.213,Z 1060.105,A -85,B 0,C 180,E1 29693.868,E2 29693.868} C_VEL
LIN {X 0,Y 317.004,Z 1056.653,A -85,B 0,C 180,E1 29694.873,E2 29694.873} C_VEL
LIN {X 0,Y 318.172,Z 1054.889,A -85,B 0,C 180,E1 29698.661,E2 29698.661} C_VEL
LIN {X 0,Y 315.252,Z 1059.351,A -85,B 0,C 180,E1 29702.757,E2 29702.757} C_VEL
LIN {X 0,Y 257.239,Z 1113.815,A -85,B 0,C 180,E1 29708.518,E2 29708.518} C_VEL
LIN {X 0,Y 196.493,Z 1155.614,A -85,B 0,C 180,E1 29719,E2 29719} C_VEL
LIN {X 0,Y 142.095,Z 1184.445,A -85,B 0,C 180,E1 29739.687,E2 29739.687} C_VEL
LIN {X 0,Y 116.668,Z 1197.598,A -85,B 0,C 180,E1 29771.029,E2 29771.029} C_VEL
LIN {X 0,Y 114.944,Z 1199.276,A -85,B 0,C 180,E1 29793.775,E2 29793.775} C_VEL
LIN {X 0,Y 123.688,Z 1193.548,A -85,B 0,C 180,E1 29823.478,E2 29823.478} C_VEL
LIN {X 0,Y 164.304,Z 1173.454,A -85,B 0,C 180,E1 29851.253,E2 29851.253} C_VEL
LIN {X 0,Y 224.21,Z 1138.171,A -85,B 0,C 180,E1 29866.606,E2 29866.606} C_VEL
LIN {X 0,Y 285.284,Z 1089.924,A -85,B 0,C 180,E1 29874.574,E2 29874.574} C_VEL
LIN {X 0,Y 316.881,Z 1057.6,A -85,B 0,C 180,E1 29877.791,E2 29877.791} C_VEL
LIN {X 0,Y 318.452,Z 1054.916,A -85,B 0,C 180,E1 29881.338,E2 29881.338} C_VEL
LIN {X 0,Y 315.469,Z 1059.024,A -85,B 0,C 180,E1 29885.958,E2 29885.958} C_VEL
LIN {X 0,Y 259.21,Z 1111.31,A -85,B 0,C 180,E1 29891.506,E2 29891.506} C_VEL
LIN {X 0,Y 198.312,Z 1152.168,A -85,B 0,C 180,E1 29901.787,E2 29901.787} C_VEL
LIN {X 0,Y 147.664,Z 1177.695,A -85,B 0,C 180,E1 29919.633,E2 29919.633} C_VEL
LIN {X 0,Y 117.703,Z 1190.781,A -85,B 0,C 180,E1 29951.218,E2 29951.218} C_VEL
LIN {X 0,Y 115.331,Z 1192.171,A -85,B 0,C 180,E1 29973.777,E2 29973.777} C_VEL
LIN {X 0,Y 128.571,Z 1185.895,A -85,B 0,C 180,E1 30006.148,E2 30006.148} C_VEL
LIN {X 0,Y 142.409,Z 1179.823,A -85,B 0,C 180,E1 30017.294,E2 30017.294} C_VEL
LIN {X 0,Y 156.874,Z 1171.584,A -85,B 0,C 180,E1 30029.34,E2 30029.34} C_VEL
LIN {X 0,Y 216.417,Z 1139.944,A -85,B 0,C 180,E1 30044.489,E2 30044.489} C_VEL
LIN {X 0,Y 278.485,Z 1094.155,A -85,B 0,C 180,E1 30052.394,E2 30052.394} C_VEL
LIN {X 0,Y 311.668,Z 1062.221,A -85,B 0,C 180,E1 30055.366,E2 30055.366} C_VEL
LIN {X 0,Y 312.758,Z 1060.852,A -85,B 0,C 180,E1 30058.638,E2 30058.638} C_VEL
LIN {X 0,Y 309.908,Z 1064.406,A -85,B 0,C 180,E1 30061.637,E2 30061.637} C_VEL
LIN {X 0,Y 250.396,Z 1117.86,A -85,B 0,C 180,E1 30067.34,E2 30067.34} C_VEL
LIN {X 0,Y 187.492,Z 1158.924,A -85,B 0,C 180,E1 30078.108,E2 30078.108} C_VEL
LIN {X 0,Y 134.514,Z 1185.246,A -85,B 0,C 180,E1 30098.444,E2 30098.444} C_VEL
LIN {X 0,Y 108.972,Z 1197.346,A -85,B 0,C 180,E1 30129.632,E2 30129.632} C_VEL
LIN {X 0,Y 106.923,Z 1199.027,A -85,B 0,C 180,E1 30154.058,E2 30154.058} C_VEL
LIN {X 0,Y 116.846,Z 1193.291,A -85,B 0,C 180,E1 30185.726,E2 30185.726} C_VEL
LIN {X 0,Y 160.425,Z 1173.191,A -85,B 0,C 180,E1 30213.89,E2 30213.89} C_VEL
LIN {X 0,Y 221.104,Z 1138.751,A -85,B 0,C 180,E1 30228.502,E2 30228.502} C_VEL
LIN {X 0,Y 282.777,Z 1091.254,A -85,B 0,C 180,E1 30236.08,E2 30236.08} C_VEL
LIN {X 0,Y 311.685,Z 1062.825,A -85,B 0,C 180,E1 30238.576,E2 30238.576} C_VEL
LIN {X 0,Y 313.022,Z 1060.891,A -85,B 0,C 180,E1 30241.361,E2 30241.361} C_VEL
LIN {X 0,Y 310.627,Z 1063.639,A -85,B 0,C 180,E1 30244.8,E2 30244.8} C_VEL
LIN {X 0,Y 252.35,Z 1115.536,A -85,B 0,C 180,E1 30250.32,E2 30250.32} C_VEL
LIN {X 0,Y 190.379,Z 1155.107,A -85,B 0,C 180,E1 30260.627,E2 30260.627} C_VEL
LIN {X 0,Y 137.869,Z 1179.809,A -85,B 0,C 180,E1 30279.658,E2 30279.658} C_VEL
LIN {X 0,Y 110.054,Z 1191.031,A -85,B 0,C 180,E1 30309.858,E2 30309.858} C_VEL
LIN {X 0,Y 107.338,Z 1192.418,A -85,B 0,C 180,E1 30334.059,E2 30334.059} C_VEL
LIN {X 0,Y 122.055,Z 1186.147,A -85,B 0,C 180,E1 30368.416,E2 30368.416} C_VEL
LIN {X 0,Y 156.874,Z 1171.584,A -85,B 0,C 180,E1 30389.34,E2 30389.34} C_VEL
LIN {X 0,Y 176.106,Z 1161.088,A -85,B 0,C 180,E1 30399.01,E2 30399.01} C_VEL
LIN {X 0,Y 238.731,Z 1124.453,A -85,B 0,C 180,E1 30409.959,E2 30409.959} C_VEL
LIN {X 0,Y 298.117,Z 1075.709,A -85,B 0,C 180,E1 30415.752,E2 30415.752} C_VEL
LIN {X 0,Y 306.425,Z 1067.311,A -85,B 0,C 180,E1 30416.672,E2 30416.672} C_VEL
LIN {X 0,Y 305.755,Z 1068.238,A -85,B 0,C 180,E1 30420.385,E2 30420.385} C_VEL
LIN {X 0,Y 245.744,Z 1120.351,A -85,B 0,C 180,E1 30425.857,E2 30425.857} C_VEL
LIN {X 0,Y 181.788,Z 1160.445,A -85,B 0,C 180,E1 30436.375,E2 30436.375} C_VEL
LIN {X 0,Y 125.326,Z 1186.782,A -85,B 0,C 180,E1 30458.126,E2 30458.126} C_VEL
LIN {X 0,Y 101.368,Z 1197.094,A -85,B 0,C 180,E1 30488.027,E2 30488.027} C_VEL
LIN {X 0,Y 98.895,Z 1198.779,A -85,B 0,C 180,E1 30514.389,E2 30514.389} C_VEL
LIN {X 0,Y 110.206,Z 1193.035,A -85,B 0,C 180,E1 30548.25,E2 30548.25} C_VEL
LIN {X 0,Y 156.914,Z 1172.932,A -85,B 0,C 180,E1 30576.641,E2 30576.641} C_VEL
LIN {X 0,Y 220.026,Z 1138.2,A -85,B 0,C 180,E1 30590.718,E2 30590.718} C_VEL
LIN {X 0,Y 283.216,Z 1090.187,A -85,B 0,C 180,E1 30597.853,E2 30597.853} C_VEL
LIN {X 0,Y 306.604,Z 1067.599,A -85,B 0,C 180,E1 30599.971,E2 30599.971} C_VEL
LIN {X 0,Y 305.689,Z 1068.411,A -85,B 0,C 180,E1 30603.623,E2 30603.623} C_VEL
LIN {X 0,Y 247.337,Z 1118.503,A -85,B 0,C 180,E1 30608.891,E2 30608.891} C_VEL
LIN {X 0,Y 184.389,Z 1157.069,A -85,B 0,C 180,E1 30618.961,E2 30618.961} C_VEL
LIN {X 0,Y 128.06,Z 1181.923,A -85,B 0,C 180,E1 30639.68,E2 30639.68} C_VEL
LIN {X 0,Y 102.492,Z 1191.281,A -85,B 0,C 180,E1 30668.299,E2 30668.299} C_VEL
LIN {X 0,Y 99.363,Z 1192.56,A -85,B 0,C 180,E1 30697.549,E2 30697.549} C_VEL
LIN {X 0,Y 119.557,Z 1184.948,A -85,B 0,C 180,E1 30734.248,E2 30734.248} C_VEL
LIN {X 0,Y 171.879,Z 1163.128,A -85,B 0,C 180,E1 30757.898,E2 30757.898} C_VEL
LIN {X 0,Y 176.106,Z 1161.088,A -85,B 0,C 180,E1 30759.01,E2 30759.01} C_VEL
LIN {X 0,Y 198.391,Z 1148.551,A -85,B 0,C 180,E1 30766.558,E2 30766.558} C_VEL
LIN {X 0,Y 262.811,Z 1106.141,A -85,B 0,C 180,E1 30774.529,E2 30774.529} C_VEL
LIN {X 0,Y 301.182,Z 1072.568,A -85,B 0,C 180,E1 30777.92,E2 30777.92} C_VEL
LIN {X 0,Y 300.262,Z 1073.59,A -85,B 0,C 180,E1 30779.207,E2 30779.207} C_VEL
LIN {X 0,Y 239.315,Z 1124.241,A -85,B 0,C 180,E1 30784.563,E2 30784.563} C_VEL
LIN {X 0,Y 174.611,Z 1162.722,A -85,B 0,C 180,E1 30794.885,E2 30794.885} C_VEL
LIN {X 0,Y 120.338,Z 1186.521,A -85,B 0,C 180,E1 30814.989,E2 30814.989} C_VEL
LIN {X 0,Y 93.828,Z 1196.841,A -85,B 0,C 180,E1 30846.157,E2 30846.157} C_VEL
LIN {X 0,Y 90.863,Z 1198.53,A -85,B 0,C 180,E1 30874.777,E2 30874.777} C_VEL
LIN {X 0,Y 103.813,Z 1192.779,A -85,B 0,C 180,E1 30911.088,E2 30911.088} C_VEL
LIN {X 0,Y 154.984,Z 1172.128,A -85,B 0,C 180,E1 30939.893,E2 30939.893} C_VEL
LIN {X 0,Y 221.414,Z 1136.323,A -85,B 0,C 180,E1 30953.248,E2 30953.248} C_VEL
LIN {X 0,Y 284.856,Z 1088.319,A -85,B 0,C 180,E1 30959.688,E2 30959.688} C_VEL
LIN {X 0,Y 301.444,Z 1072.674,A -85,B 0,C 180,E1 30960.984,E2 30960.984} C_VEL
LIN {X 0,Y 300.334,Z 1073.742,A -85,B 0,C 180,E1 30962.443,E2 30962.443} C_VEL
LIN {X 0,Y 239.559,Z 1123.503,A -85,B 0,C 180,E1 30967.744,E2 30967.744} C_VEL
LIN {X 0,Y 175.709,Z 1160.356,A -85,B 0,C 180,E1 30977.81,E2 30977.81} C_VEL
LIN {X 0,Y 119.173,Z 1183.471,A -85,B 0,C 180,E1 30999.057,E2 30999.057} C_VEL
LIN {X 0,Y 92.251,Z 1192.489,A -85,B 0,C 180,E1 31035.734,E2 31035.734} C_VEL
LIN {X 0,Y 92.244,Z 1192.461,A -85,B 0,C 180,E1 31064.286,E2 31064.286} C_VEL
LIN {X 0,Y 119.291,Z 1183.37,A -85,B 0,C 180,E1 31100.98,E2 31100.98} C_VEL
LIN {X 0,Y 178.347,Z 1159.006,A -85,B 0,C 180,E1 31122.723,E2 31122.723} C_VEL
LIN {X 0,Y 198.391,Z 1148.551,A -85,B 0,C 180,E1 31126.558,E2 31126.558} C_VEL
LIN {X 0,Y 222.7,Z 1133.875,A -85,B 0,C 180,E1 31132.372,E2 31132.372} C_VEL
LIN {X 0,Y 285.361,Z 1087.365,A -85,B 0,C 180,E1 31138.071,E2 31138.071} C_VEL
LIN {X 0,Y 285.285,Z 1087.461,A -85,B 0,C 180,E1 31138.602,E2 31138.602} C_VEL
LIN {X 0,Y 220.605,Z 1135.875,A -85,B 0,C 180,E1 31144.552,E2 31144.552} C_VEL
LIN {X 0,Y 154.222,Z 1170.907,A -85,B 0,C 180,E1 31156.495,E2 31156.495} C_VEL
LIN {X 0,Y 100.406,Z 1191.598,A -85,B 0,C 180,E1 31182.984,E2 31182.984} C_VEL
LIN {X 0,Y 83.627,Z 1197.715,A -85,B 0,C 180,E1 31214.205,E2 31214.205} C_VEL
LIN {X 0,Y 82.832,Z 1198.281,A -85,B 0,C 180,E1 31235.242,E2 31235.242} C_VEL
LIN {X 0,Y 97.689,Z 1192.522,A -85,B 0,C 180,E1 31274.301,E2 31274.301} C_VEL
LIN {X 0,Y 151.028,Z 1172.41,A -85,B 0,C 180,E1 31302.52,E2 31302.52} C_VEL
LIN {X 0,Y 218.748,Z 1137.164,A -85,B 0,C 180,E1 31315.202,E2 31315.202} C_VEL
LIN {X 0,Y 283.583,Z 1089.178,A -85,B 0,C 180,E1 31321.277,E2 31321.277} C_VEL
LIN {X 0,Y 286.583,Z 1086.544,A -85,B 0,C 180,E1 31321.486,E2 31321.486} C_VEL
LIN {X 0,Y 223.638,Z 1133.481,A -85,B 0,C 180,E1 31327.401,E2 31327.401} C_VEL
LIN {X 0,Y 156.444,Z 1168.073,A -85,B 0,C 180,E1 31339.086,E2 31339.086} C_VEL
LIN {X 0,Y 103.923,Z 1186.968,A -85,B 0,C 180,E1 31363.156,E2 31363.156} C_VEL
LIN {X 0,Y 83.26,Z 1193.174,A -85,B 0,C 180,E1 31404.785,E2 31404.785} C_VEL
LIN {X 0,Y 87.626,Z 1191.754,A -85,B 0,C 180,E1 31435.648,E2 31435.648} C_VEL
LIN {X 0,Y 129.108,Z 1178.617,A -85,B 0,C 180,E1 31471.772,E2 31471.772} C_VEL
LIN {X 0,Y 193.528,Z 1150.519,A -85,B 0,C 180,E1 31488.406,E2 31488.406} C_VEL
LIN {X 0,Y 222.7,Z 1133.875,A -85,B 0,C 180,E1 31492.372,E2 31492.372} C_VEL
LIN {X 0,Y 247.661,Z 1117.061,A -85,B 0,C 180,E1 31496.966,E2 31496.966} C_VEL
LIN {X 0,Y 262.843,Z 1105.895,A -85,B 0,C 180,E1 31498.472,E2 31498.472} C_VEL
LIN {X 0,Y 197.926,Z 1148.443,A -85,B 0,C 180,E1 31505.101,E2 31505.101} C_VEL
LIN {X 0,Y 129.49,Z 1179.64,A -85,B 0,C 180,E1 31520.253,E2 31520.253} C_VEL
LIN {X 0,Y 84.651,Z 1194.541,A -85,B 0,C 180,E1 31551.156,E2 31551.156} C_VEL
LIN {X 0,Y 74.926,Z 1198.029,A -85,B 0,C 180,E1 31584.18,E2 31584.18} C_VEL
LIN {X 0,Y 80.378,Z 1195.903,A -85,B 0,C 180,E1 31621.605,E2 31621.605} C_VEL
LIN {X 0,Y 126.084,Z 1181.019,A -85,B 0,C 180,E1 31658.551,E2 31658.551} C_VEL
LIN {X 0,Y 194.209,Z 1150.612,A -85,B 0,C 180,E1 31674.413,E2 31674.413} C_VEL
LIN {X 0,Y 260.785,Z 1107.729,A -85,B 0,C 180,E1 31681.337,E2 31681.337} C_VEL
LIN {X 0,Y 263.126,Z 1105.9,A -85,B 0,C 180,E1 31681.722,E2 31681.722} C_VEL
LIN {X 0,Y 197.275,Z 1148.134,A -85,B 0,C 180,E1 31688.419,E2 31688.419} C_VEL
LIN {X 0,Y 131.478,Z 1176.816,A -85,B 0,C 180,E1 31702.686,E2 31702.686} C_VEL
LIN {X 0,Y 86.053,Z 1190.503,A -85,B 0,C 180,E1 31732.364,E2 31732.364} C_VEL
LIN {X 0,Y 75.259,Z 1193.422,A -85,B 0,C 180,E1 31764.229,E2 31764.229} C_VEL
LIN {X 0,Y 80.377,Z 1192.005,A -85,B 0,C 180,E1 31798.156,E2 31798.156} C_VEL
LIN {X 0,Y 125.434,Z 1178.871,A -85,B 0,C 180,E1 31835.078,E2 31835.078} C_VEL
LIN {X 0,Y 192.042,Z 1150.785,A -85,B 0,C 180,E1 31850.815,E2 31850.815} C_VEL
LIN {X 0,Y 247.661,Z 1117.061,A -85,B 0,C 180,E1 31856.966,E2 31856.966} C_VEL
LIN {X 0,Y 243.299,Z 1120.138,A -85,B 0,C 180,E1 31858.082,E2 31858.082} C_VEL
LIN {X 0,Y 229.474,Z 1129.31,A -85,B 0,C 180,E1 31859.312,E2 31859.312} C_VEL
LIN {X 0,Y 160.89,Z 1165.89,A -85,B 0,C 180,E1 31868.191,E2 31868.191} C_VEL
LIN {X 0,Y 96.566,Z 1189.114,A -85,B 0,C 180,E1 31890.243,E2 31890.243} C_VEL
LIN {X 0,Y 68.107,Z 1197.212,A -85,B 0,C 180,E1 31930.475,E2 31930.475} C_VEL
LIN {X 0,Y 66.78,Z 1197.783,A -85,B 0,C 180,E1 31956.507,E2 31956.507} C_VEL
LIN {X 0,Y 86.566,Z 1192.01,A -85,B 0,C 180,E1 32002.014,E2 32002.014} C_VEL
LIN {X 0,Y 146.841,Z 1171.883,A -85,B 0,C 180,E1 32028.817,E2 32028.817} C_VEL
LIN {X 0,Y 217.988,Z 1136.624,A -85,B 0,C 180,E1 32039.626,E2 32039.626} C_VEL
LIN {X 0,Y 237.987,Z 1123.995,A -85,B 0,C 180,E1 32041.79,E2 32041.79} C_VEL
LIN {X 0,Y 168.109,Z 1161.837,A -85,B 0,C 180,E1 32050.129,E2 32050.129} C_VEL
LIN {X 0,Y 104.206,Z 1184.539,A -85,B 0,C 180,E1 32069.187,E2 32069.187} C_VEL
LIN {X 0,Y 69.013,Z 1193.237,A -85,B 0,C 180,E1 32110.768,E2 32110.768} C_VEL
LIN {X 0,Y 69.016,Z 1193.211,A -85,B 0,C 180,E1 32149.258,E2 32149.258} C_VEL
LIN {X 0,Y 104.232,Z 1184.466,A -85,B 0,C 180,E1 32190.822,E2 32190.822} C_VEL
LIN {X 0,Y 168.45,Z 1161.565,A -85,B 0,C 180,E1 32209.91,E2 32209.91} C_VEL
LIN {X 0,Y 237.826,Z 1123.901,A -85,B 0,C 180,E1 32218.106,E2 32218.106} C_VEL
LIN {X 0,Y 229.474,Z 1129.31,A -85,B 0,C 180,E1 32219.312,E2 32219.312} C_VEL
LIN {X 0,Y 209.482,Z 1141.116,A -85,B 0,C 180,E1 32217.723,E2 32217.723} C_VEL
LIN {X 0,Y 141.837,Z 1171.847,A -85,B 0,C 180,E1 32207.986,E2 32207.986} C_VEL
LIN {X 0,Y 78.626,Z 1189.976,A -85,B 0,C 180,E1 32180.506,E2 32180.506} C_VEL
LIN {X 0,Y 59.344,Z 1193.908,A -85,B 0,C 180,E1 32137.356,E2 32137.356} C_VEL
LIN {X 0,Y 70.644,Z 1191.628,A -85,B 0,C 180,E1 32088.571,E2 32088.571} C_VEL
LIN {X 0,Y 126.023,Z 1177.329,A -85,B 0,C 180,E1 32055.726,E2 32055.726} C_VEL
LIN {X 0,Y 197.481,Z 1147.659,A -85,B 0,C 180,E1 32043.41,E2 32043.41} C_VEL
LIN {X 0,Y 213.523,Z 1139.007,A -85,B 0,C 180,E1 32041.429,E2 32041.429} C_VEL
LIN {X 0,Y 140.773,Z 1173.438,A -85,B 0,C 180,E1 32031.09,E2 32031.09} C_VEL
LIN {X 0,Y 81.698,Z 1191.754,A -85,B 0,C 180,E1 32006.629,E2 32006.629} C_VEL
LIN {X 0,Y 58.763,Z 1197.534,A -85,B 0,C 180,E1 31957.399,E2 31957.399} C_VEL
LIN {X 0,Y 65.217,Z 1195.83,A -85,B 0,C 180,E1 31914.439,E2 31914.439} C_VEL
LIN {X 0,Y 117.811,Z 1181.456,A -85,B 0,C 180,E1 31875.081,E2 31875.081} C_VEL
LIN {X 0,Y 189.612,Z 1151.889,A -85,B 0,C 180,E1 31861.071,E2 31861.071} C_VEL
LIN {X 0,Y 213.781,Z 1138.69,A -85,B 0,C 180,E1 31858.539,E2 31858.539} C_VEL
LIN {X 0,Y 209.482,Z 1141.116,A -85,B 0,C 180,E1 31857.723,E2 31857.723} C_VEL
LIN {X 0,Y 177.851,Z 1157.049,A -85,B 0,C 180,E1 31856.941,E2 31856.941} C_VEL
LIN {X 0,Y 108.061,Z 1182.145,A -85,B 0,C 180,E1 31843.396,E2 31843.396} C_VEL
LIN {X 0,Y 60.001,Z 1192.757,A -85,B 0,C 180,E1 31809.207,E2 31809.207} C_VEL
LIN {X 0,Y 51.339,Z 1194.166,A -85,B 0,C 180,E1 31761.524,E2 31761.524} C_VEL
LIN {X 0,Y 86.276,Z 1187.704,A -85,B 0,C 180,E1 31705.977,E2 31705.977} C_VEL
LIN {X 0,Y 156.244,Z 1166.34,A -85,B 0,C 180,E1 31685.86,E2 31685.86} C_VEL
LIN {X 0,Y 189.616,Z 1151.776,A -85,B 0,C 180,E1 31681.522,E2 31681.522} C_VEL
LIN {X 0,Y 115.836,Z 1181.268,A -85,B 0,C 180,E1 31669.04,E2 31669.04} C_VEL
LIN {X 0,Y 58.657,Z 1195.595,A -85,B 0,C 180,E1 31630.248,E2 31630.248} C_VEL
LIN {X 0,Y 50.876,Z 1197.28,A -85,B 0,C 180,E1 31581.411,E2 31581.411} C_VEL
LIN {X 0,Y 77.459,Z 1191.445,A -85,B 0,C 180,E1 31528.211,E2 31528.211} C_VEL
LIN {X 0,Y 144.532,Z 1171.238,A -85,B 0,C 180,E1 31504.512,E2 31504.512} C_VEL
LIN {X 0,Y 189.673,Z 1151.582,A -85,B 0,C 180,E1 31498.198,E2 31498.198} C_VEL
LIN {X 0,Y 177.851,Z 1157.049,A -85,B 0,C 180,E1 31496.941,E2 31496.941} C_VEL
LIN {X 0,Y 145.139,Z 1170.313,A -85,B 0,C 180,E1 31495.59,E2 31495.59} C_VEL
LIN {X 0,Y 75.337,Z 1189.327,A -85,B 0,C 180,E1 31474.964,E2 31474.964} C_VEL
LIN {X 0,Y 43.426,Z 1194.406,A -85,B 0,C 180,E1 31420.076,E2 31420.076} C_VEL
LIN {X 0,Y 55.718,Z 1192.756,A -85,B 0,C 180,E1 31362.706,E2 31362.706} C_VEL
LIN {X 0,Y 118.996,Z 1178.957,A -85,B 0,C 180,E1 31329.051,E2 31329.051} C_VEL
LIN {X 0,Y 165.213,Z 1162.756,A -85,B 0,C 180,E1 31321.557,E2 31321.557} C_VEL
LIN {X 0,Y 94.222,Z 1186.576,A -85,B 0,C 180,E1 31307.073,E2 31307.073} C_VEL
LIN {X 0,Y 45.796,Z 1196.477,A -85,B 0,C 180,E1 31259.762,E2 31259.762} C_VEL
LIN {X 0,Y 42.888,Z 1197.03,A -85,B 0,C 180,E1 31219.796,E2 31219.796} C_VEL
LIN {X 0,Y 73.87,Z 1191.187,A -85,B 0,C 180,E1 31162.477,E2 31162.477} C_VEL
LIN {X 0,Y 144.114,Z 1170.975,A -85,B 0,C 180,E1 31141.166,E2 31141.166} C_VEL
LIN {X 0,Y 165.398,Z 1162.558,A -85,B 0,C 180,E1 31138.423,E2 31138.423} C_VEL
LIN {X 0,Y 145.139,Z 1170.313,A -85,B 0,C 180,E1 31135.59,E2 31135.59} C_VEL
LIN {X 0,Y 111.469,Z 1180.882,A -85,B 0,C 180,E1 31133.578,E2 31133.578} C_VEL
LIN {X 0,Y 48.492,Z 1193.259,A -85,B 0,C 180,E1 31101.457,E2 31101.457} C_VEL
LIN {X 0,Y 35.503,Z 1194.663,A -85,B 0,C 180,E1 31037.693,E2 31037.693} C_VEL
LIN {X 0,Y 75.955,Z 1188.986,A -85,B 0,C 180,E1 30977.319,E2 30977.319} C_VEL
LIN {X 0,Y 139.31,Z 1172.584,A -85,B 0,C 180,E1 30961.464,E2 30961.464} C_VEL
LIN {X 0,Y 71.077,Z 1190.981,A -85,B 0,C 180,E1 30943.722,E2 30943.722} C_VEL
LIN {X 0,Y 34.857,Z 1196.785,A -85,B 0,C 180,E1 30882.539,E2 30882.539} C_VEL
LIN {X 0,Y 38.952,Z 1196.203,A -85,B 0,C 180,E1 30834.241,E2 30834.241} C_VEL
LIN {X 0,Y 91.907,Z 1186.435,A -85,B 0,C 180,E1 30788.03,E2 30788.03} C_VEL
LIN {X 0,Y 139.224,Z 1172.501,A -85,B 0,C 180,E1 30778.448,E2 30778.448} C_VEL
LIN {X 0,Y 111.469,Z 1180.882,A -85,B 0,C 180,E1 30773.578,E2 30773.578} C_VEL
LIN {X 0,Y 77.291,Z 1188.55,A -85,B 0,C 180,E1 30769.96,E2 30769.96} C_VEL
LIN {X 0,Y 27.716,Z 1194.903,A -85,B 0,C 180,E1 30705.91,E2 30705.91} C_VEL
LIN {X 0,Y 43.877,Z 1193.534,A -85,B 0,C 180,E1 30630.262,E2 30630.262} C_VEL
LIN {X 0,Y 113.769,Z 1180.493,A -85,B 0,C 180,E1 30601.618,E2 30601.618} C_VEL
LIN {X 0,Y 42.861,Z 1194.832,A -85,B 0,C 180,E1 30572.152,E2 30572.152} C_VEL
LIN {X 0,Y 27.092,Z 1196.53,A -85,B 0,C 180,E1 30493.714,E2 30493.714} C_VEL
LIN {X 0,Y 69.219,Z 1190.669,A -85,B 0,C 180,E1 30429.559,E2 30429.559} C_VEL
LIN {X 0,Y 113.805,Z 1180.401,A -85,B 0,C 180,E1 30418.273,E2 30418.273} C_VEL
LIN {X 0,Y 77.291,Z 1188.55,A -85,B 0,C 180,E1 30409.96,E2 30409.96} C_VEL
LIN {X 0,Y 42.966,Z 1193.456,A -85,B 0,C 180,E1 30401.928,E2 30401.928} C_VEL
LIN {X 0,Y 20.055,Z 1195.161,A -85,B 0,C 180,E1 30307.831,E2 30307.831} C_VEL
LIN {X 0,Y 75.998,Z 1188.99,A -85,B 0,C 180,E1 30244.026,E2 30244.026} C_VEL
LIN {X 0,Y 83.405,Z 1187.632,A -85,B 0,C 180,E1 30240.973,E2 30240.973} C_VEL
LIN {X 0,Y 27.373,Z 1195.72,A -85,B 0,C 180,E1 30206.146,E2 30206.146} C_VEL
LIN {X 0,Y 19.443,Z 1196.279,A -85,B 0,C 180,E1 30126.997,E2 30126.997} C_VEL
LIN {X 0,Y 68.33,Z 1190.411,A -85,B 0,C 180,E1 30062.626,E2 30062.626} C_VEL
LIN {X 0,Y 83.491,Z 1187.503,A -85,B 0,C 180,E1 30057.7,E2 30057.7} C_VEL
LIN {X 0,Y 42.966,Z 1193.456,A -85,B 0,C 180,E1 30041.928,E2 30041.928} C_VEL
LIN {X 0,Y 11.855,Z 1195.402,A -85,B 0,C 180,E1 29997.385,E2 29997.385} C_VEL
LIN {X 0,Y 38.342,Z 1194.036,A -85,B 0,C 180,E1 29888.734,E2 29888.734} C_VEL
LIN {X 0,Y 56.59,Z 1192.095,A -85,B 0,C 180,E1 29881.638,E2 29881.638} C_VEL
LIN {X 0,Y 12.317,Z 1196.034,A -85,B 0,C 180,E1 29827.908,E2 29827.908} C_VEL
LIN {X 0,Y 23.839,Z 1195.446,A -85,B 0,C 180,E1 29717.285,E2 29717.285} C_VEL
LIN {X 0,Y 53.158,Z 1192.425,A -85,B 0,C 180,E1 29697.171,E2 29697.171} C_VEL
LIN {X 0,Y 11.855,Z 1195.402,A -85,B 0,C 180,E1 29637.385,E2 29637.385} C_VEL
LIN {X 0,Y 16.464,Z 1195.508,A -85,B 0,C 180,E1 29522.773,E2 29522.773} C_VEL
LIN {X 0,Y 18.976,Z 1195.465,A -85,B 0,C 180,E1 29520.987,E2 29520.987} C_VEL
LIN {X 0,Y 7.778,Z 1195.778,A -85,B 0,C 180,E1 29352.366,E2 29352.366} C_VEL
LIN {X 0,Y 19.048,Z 1195.454,A -85,B 0,C 180,E1 29339.035,E2 29339.035} C_VEL
LIN {X 0,Y 16.464,Z 1195.508,A -85,B 0,C 180,E1 29162.773,E2 29162.773} C_VEL
LIN {X 0,Y 18.449,Z 1197.507,A -85,B 0,C 180,E1 29161.321,E2 29161.321} C_VEL
LIN {X 0,Y 18.449,Z 1215,A -85,B 0,C 180,E1 29161.321,E2 29161.321} C_VEL
LIN {X 0,Y 18.449,Z 1215,A -85,B 0,C 180,E1 29161.321,E2 29161.321}

QRS_NEXT_CUT()
PTP {E1 29337.24,E2 29337.24}
PTP {X 0,Y 759.899,A -85,B 0,C 180,E1 29337.24,E2 29337.24,E3 0,E4 0,E5 0,E6 0}
QRS_SPEED_INIT()
LIN {X 0,Y 759.899,Z 1215,A -85,B 0,C 180,E1 29337.24,E2 29337.24,E3 0,E4 0,E5 0,E6 0} C_VEL
LIN {X 0,Y 759.899,Z 319.643,A -85,B 0,C 180,E1 29337.24,E2 29337.24} C_VEL
LIN {X 0,Y 759.899,Z 311.567,A -85,B 0,C 180,E1 29337.24,E2 29337.24} C_VEL
LIN {X 0,Y 759.888,Z 309.567,A -85,B 0,C 180,E1 29337.089,E2 29337.089} C_VEL
LIN {X 0,Y 759.912,Z 309.576,A -85,B 0,C 180,E1 29334.261,E2 29334.261} C_VEL
LIN {X 0,Y 759.916,Z 309.563,A -85,B 0,C 180,E1 29331.22,E2 29331.22} C_VEL
LIN {X 0,Y 759.914,Z 309.576,A -85,B 0,C 180,E1 29328.155,E2 29328.155} C_VEL
LIN {X 0,Y 759.911,Z 309.564,A -85,B 0,C 180,E1 29325.133,E2 29325.133} C_VEL
LIN {X 0,Y 759.911,Z 309.575,A -85,B 0,C 180,E1 29322.047,E2 29322.047} C_VEL
LIN {X 0,Y 759.898,Z 309.565,A -85,B 0,C 180,E1 29319.103,E2 29319.103} C_VEL
LIN {X 0,Y 759.916,Z 309.576,A -85,B 0,C 180,E1 29316.092,E2 29316.092} C_VEL
LIN {X 0,Y 759.873,Z 309.57,A -85,B 0,C 180,E1 29313.312,E2 29313.312} C_VEL
LIN {X 0,Y 759.908,Z 309.566,A -85,B 0,C 180,E1 29310.52,E2 29310.52} C_VEL
LIN {X 0,Y 759.88,Z 309.573,A -85,B 0,C 180,E1 29307.618,E2 29307.618} C_VEL
LIN {X 0,Y 759.874,Z 309.569,A -85,B 0,C 180,E1 29304.898,E2 29304.898} C_VEL
LIN {X 0,Y 759.914,Z 309.574,A -85,B 0,C 180,E1 29301.99,E2 29301.99} C_VEL
LIN {X 0,Y 759.857,Z 309.572,A -85,B 0,C 180,E1 29299.256,E2 29299.256} C_VEL
LIN {X 0,Y 759.867,Z 309.57,A -85,B 0,C 180,E1 29296.692,E2 29296.692} C_VEL
LIN {X 0,Y 759.915,Z 309.574,A -85,B 0,C 180,E1 29293.749,E2 29293.749} C_VEL
LIN {X 0,Y 759.915,Z 309.82,A -85,B 0,C 180,E1 29291.976,E2 29291.976} C_VEL
LIN {X 0,Y 759.917,Z 320.268,A -85,B 0,C 180,E1 29291.295,E2 29291.295} C_VEL
LIN {X 0,Y 759.891,Z 362.671,A -85,B 0,C 180,E1 29288.713,E2 29288.713} C_VEL
LIN {X 0,Y 759.879,Z 396.77,A -85,B 0,C 180,E1 29286.719,E2 29286.719} C_VEL
LIN {X 0,Y 759.916,Z 616.143,A -85,B 0,C 180,E1 29284.217,E2 29284.217} C_VEL
LIN {X 0,Y 759.915,Z 828.9,A -85,B 0,C 180,E1 29281.845,E2 29281.845} C_VEL
LIN {X 0,Y 759.913,Z 848.684,A -85,B 0,C 180,E1 29281.54,E2 29281.54} C_VEL
LIN {X 0,Y 759.911,Z 872.955,A -85,B 0,C 180,E1 29281.05,E2 29281.05} C_VEL
LIN {X 0,Y 759.913,Z 896.954,A -85,B 0,C 180,E1 29280.414,E2 29280.414} C_VEL
LIN {X 0,Y 759.916,Z 915.69,A -85,B 0,C 180,E1 29279.826,E2 29279.826} C_VEL
LIN {X 0,Y 759.917,Z 934.841,A -85,B 0,C 180,E1 29279.133,E2 29279.133} C_VEL
LIN {X 0,Y 759.915,Z 954.435,A -85,B 0,C 180,E1 29278.325,E2 29278.325} C_VEL
LIN {X 0,Y 759.91,Z 978.395,A -85,B 0,C 180,E1 29277.191,E2 29277.191} C_VEL
LIN {X 0,Y 759.917,Z 998.211,A -85,B 0,C 180,E1 29276.112,E2 29276.112} C_VEL
LIN {X 0,Y 759.902,Z 1016.814,A -85,B 0,C 180,E1 29274.985,E2 29274.985} C_VEL
LIN {X 0,Y 759.905,Z 1038.621,A -85,B 0,C 180,E1 29273.491,E2 29273.491} C_VEL
LIN {X 0,Y 759.916,Z 1055.534,A -85,B 0,C 180,E1 29272.187,E2 29272.187} C_VEL
LIN {X 0,Y 759.918,Z 1074.324,A -85,B 0,C 180,E1 29270.568,E2 29270.568} C_VEL
LIN {X 0,Y 759.902,Z 1089.145,A -85,B 0,C 180,E1 29269.125,E2 29269.125} C_VEL
LIN {X 0,Y 759.909,Z 1103.828,A -85,B 0,C 180,E1 29267.537,E2 29267.537} C_VEL
LIN {X 0,Y 759.895,Z 1118.432,A -85,B 0,C 180,E1 29265.727,E2 29265.727} C_VEL
LIN {X 0,Y 759.914,Z 1128.969,A -85,B 0,C 180,E1 29264.244,E2 29264.244} C_VEL
LIN {X 0,Y 759.917,Z 1139.18,A -85,B 0,C 180,E1 29262.616,E2 29262.616} C_VEL
LIN {X 0,Y 759.893,Z 1149.873,A -85,B 0,C 180,E1 29260.601,E2 29260.601} C_VEL
LIN {X 0,Y 759.911,Z 1156.887,A -85,B 0,C 180,E1 29259.008,E2 29259.008} C_VEL
LIN {X 0,Y 759.9,Z 1162.494,A -85,B 0,C 180,E1 29257.485,E2 29257.485} C_VEL
LIN {X 0,Y 759.892,Z 1167.442,A -85,B 0,C 180,E1 29255.815,E2 29255.815} C_VEL
LIN {X 0,Y 759.913,Z 1171.769,A -85,B 0,C 180,E1 29253.772,E2 29253.772} C_VEL
LIN {X 0,Y 759.914,Z 1173.964,A -85,B 0,C 180,E1 29252.036,E2 29252.036} C_VEL
LIN {X 0,Y 759.891,Z 1174.881,A -85,B 0,C 180,E1 29250.377,E2 29250.377} C_VEL
LIN {X 0,Y 759.904,Z 1174.38,A -85,B 0,C 180,E1 29248.341,E2 29248.341} C_VEL
LIN {X 0,Y 759.894,Z 1172.468,A -85,B 0,C 180,E1 29246.606,E2 29246.606} C_VEL
LIN {X 0,Y 759.904,Z 1169.601,A -85,B 0,C 180,E1 29245.018,E2 29245.018} C_VEL
LIN {X 0,Y 759.891,Z 1165.002,A -85,B 0,C 180,E1 29243.199,E2 29243.199} C_VEL
LIN {X 0,Y 759.9,Z 1158.468,A -85,B 0,C 180,E1 29241.297,E2 29241.297} C_VEL
LIN {X 0,Y 759.916,Z 1151.652,A -85,B 0,C 180,E1 29239.692,E2 29239.692} C_VEL
LIN {X 0,Y 759.905,Z 1143.98,A -85,B 0,C 180,E1 29238.155,E2 29238.155} C_VEL
LIN {X 0,Y 759.897,Z 1133.69,A -85,B 0,C 180,E1 29236.377,E2 29236.377} C_VEL
LIN {X 0,Y 759.915,Z 1121.425,A -85,B 0,C 180,E1 29234.586,E2 29234.586} C_VEL
LIN {X 0,Y 759.894,Z 1109.575,A -85,B 0,C 180,E1 29233.06,E2 29233.06} C_VEL
LIN {X 0,Y 759.907,Z 1094.692,A -85,B 0,C 180,E1 29231.353,E2 29231.353} C_VEL
LIN {X 0,Y 759.904,Z 1078.623,A -85,B 0,C 180,E1 29229.748,E2 29229.748} C_VEL
LIN {X 0,Y 759.907,Z 1062.228,A -85,B 0,C 180,E1 29228.274,E2 29228.274} C_VEL
LIN {X 0,Y 759.91,Z 1043.084,A -85,B 0,C 180,E1 29226.751,E2 29226.751} C_VEL
LIN {X 0,Y 759.908,Z 1025.733,A -85,B 0,C 180,E1 29225.514,E2 29225.514} C_VEL
LIN {X 0,Y 759.91,Z 1004.49,A -85,B 0,C 180,E1 29224.16,E2 29224.16} C_VEL
LIN {X 0,Y 759.914,Z 984.586,A -85,B 0,C 180,E1 29223.046,E2 29223.046} C_VEL
LIN {X 0,Y 759.916,Z 965.953,A -85,B 0,C 180,E1 29222.111,E2 29222.111} C_VEL
LIN {X 0,Y 759.92,Z 942.841,A -85,B 0,C 180,E1 29221.086,E2 29221.086} C_VEL
LIN {X 0,Y 759.916,Z 919.611,A -85,B 0,C 180,E1 29220.218,E2 29220.218} C_VEL
LIN {X 0,Y 759.916,Z 900.721,A -85,B 0,C 180,E1 29219.608,E2 29219.608} C_VEL
LIN {X 0,Y 759.919,Z 882.553,A -85,B 0,C 180,E1 29219.104,E2 29219.104} C_VEL
LIN {X 0,Y 759.912,Z 863.813,A -85,B 0,C 180,E1 29218.665,E2 29218.665} C_VEL
LIN {X 0,Y 759.916,Z 845.172,A -85,B 0,C 180,E1 29218.31,E2 29218.31} C_VEL
LIN {X 0,Y 759.917,Z 825.597,A -85,B 0,C 180,E1 29218.022,E2 29218.022} C_VEL
LIN {X 0,Y 759.905,Z 568.201,A -85,B 0,C 180,E1 29215.154,E2 29215.154} C_VEL
LIN {X 0,Y 759.875,Z 396.347,A -85,B 0,C 180,E1 29213.179,E2 29213.179} C_VEL
LIN {X 0,Y 759.874,Z 357.396,A -85,B 0,C 180,E1 29210.88,E2 29210.88} C_VEL
LIN {X 0,Y 759.918,Z 316.16,A -85,B 0,C 180,E1 29208.359,E2 29208.359} C_VEL
LIN {X 0,Y 759.917,Z 309.809,A -85,B 0,C 180,E1 29207.933,E2 29207.933} C_VEL
LIN {X 0,Y 759.85,Z 309.573,A -85,B 0,C 180,E1 29205.252,E2 29205.252} C_VEL
LIN {X 0,Y 759.846,Z 309.574,A -85,B 0,C 180,E1 29202.755,E2 29202.755} C_VEL
LIN {X 0,Y 759.918,Z 309.577,A -85,B 0,C 180,E1 29200.024,E2 29200.024} C_VEL
LIN {X 0,Y 759.866,Z 309.569,A -85,B 0,C 180,E1 29197.117,E2 29197.117} C_VEL
LIN {X 0,Y 759.861,Z 309.574,A -85,B 0,C 180,E1 29194.54,E2 29194.54} C_VEL
LIN {X 0,Y 759.911,Z 309.574,A -85,B 0,C 180,E1 29191.789,E2 29191.789} C_VEL
LIN {X 0,Y 759.877,Z 309.567,A -85,B 0,C 180,E1 29188.951,E2 29188.951} C_VEL
LIN {X 0,Y 759.886,Z 309.575,A -85,B 0,C 180,E1 29186.183,E2 29186.183} C_VEL
LIN {X 0,Y 759.912,Z 309.565,A -85,B 0,C 180,E1 29183.25,E2 29183.25} C_VEL
LIN {X 0,Y 759.875,Z 309.571,A -85,B 0,C 180,E1 29180.466,E2 29180.466} C_VEL
LIN {X 0,Y 759.909,Z 309.575,A -85,B 0,C 180,E1 29177.695,E2 29177.695} C_VEL
LIN {X 0,Y 759.9,Z 309.565,A -85,B 0,C 180,E1 29174.736,E2 29174.736} C_VEL
LIN {X 0,Y 759.914,Z 309.576,A -85,B 0,C 180,E1 29171.768,E2 29171.768} C_VEL
LIN {X 0,Y 759.911,Z 309.564,A -85,B 0,C 180,E1 29168.703,E2 29168.703} C_VEL
LIN {X 0,Y 759.911,Z 309.577,A -85,B 0,C 180,E1 29165.663,E2 29165.663} C_VEL
LIN {X 0,Y 759.912,Z 309.564,A -85,B 0,C 180,E1 29162.64,E2 29162.64} C_VEL
LIN {X 0,Y 759.908,Z 309.577,A -85,B 0,C 180,E1 29159.548,E2 29159.548} C_VEL
LIN {X 0,Y 759.896,Z 309.566,A -85,B 0,C 180,E1 29156.605,E2 29156.605} C_VEL
LIN {X 0,Y 759.912,Z 309.575,A -85,B 0,C 180,E1 29153.654,E2 29153.654} C_VEL
LIN {X 0,Y 759.871,Z 309.571,A -85,B 0,C 180,E1 29150.915,E2 29150.915} C_VEL
LIN {X 0,Y 759.914,Z 309.564,A -85,B 0,C 180,E1 29148.155,E2 29148.155} C_VEL
LIN {X 0,Y 759.886,Z 309.575,A -85,B 0,C 180,E1 29145.21,E2 29145.21} C_VEL
LIN {X 0,Y 759.863,Z 309.569,A -85,B 0,C 180,E1 29142.541,E2 29142.541} C_VEL
LIN {X 0,Y 759.912,Z 309.57,A -85,B 0,C 180,E1 29139.743,E2 29139.743} C_VEL
LIN {X 0,Y 759.862,Z 309.573,A -85,B 0,C 180,E1 29136.913,E2 29136.913} C_VEL
LIN {X 0,Y 759.853,Z 309.571,A -85,B 0,C 180,E1 29134.339,E2 29134.339} C_VEL
LIN {X 0,Y 759.915,Z 309.571,A -85,B 0,C 180,E1 29131.555,E2 29131.555} C_VEL
LIN {X 0,Y 759.851,Z 309.575,A -85,B 0,C 180,E1 29128.77,E2 29128.77} C_VEL
LIN {X 0,Y 759.835,Z 309.573,A -85,B 0,C 180,E1 29126.357,E2 29126.357} C_VEL
LIN {X 0,Y 759.858,Z 309.572,A -85,B 0,C 180,E1 29123.877,E2 29123.877} C_VEL
LIN {X 0,Y 759.856,Z 309.576,A -85,B 0,C 180,E1 29120.809,E2 29120.809} C_VEL
LIN {X 0,Y 759.822,Z 309.576,A -85,B 0,C 180,E1 29118.351,E2 29118.351} C_VEL
LIN {X 0,Y 759.818,Z 309.571,A -85,B 0,C 180,E1 29116.091,E2 29116.091} C_VEL
LIN {X 0,Y 759.833,Z 309.559,A -85,B 0,C 180,E1 29113.743,E2 29113.743} C_VEL
LIN {X 0,Y 759.893,Z 309.922,A -85,B 0,C 180,E1 29113.328,E2 29113.328} C_VEL
LIN {X 0,Y 759.92,Z 341.3,A -85,B 0,C 180,E1 29111.439,E2 29111.439} C_VEL
LIN {X 0,Y 759.904,Z 350.286,A -85,B 0,C 180,E1 29110.927,E2 29110.927} C_VEL
LIN {X 0,Y 759.919,Z 553.72,A -85,B 0,C 180,E1 29108.473,E2 29108.473} C_VEL
LIN {X 0,Y 759.913,Z 781.497,A -85,B 0,C 180,E1 29105.828,E2 29105.828} C_VEL
LIN {X 0,Y 759.91,Z 830.455,A -85,B 0,C 180,E1 29105.243,E2 29105.243} C_VEL
LIN {X 0,Y 759.91,Z 856.588,A -85,B 0,C 180,E1 29104.789,E2 29104.789} C_VEL
LIN {X 0,Y 759.914,Z 883.591,A -85,B 0,C 180,E1 29104.163,E2 29104.163} C_VEL
LIN {X 0,Y 759.908,Z 907.506,A -85,B 0,C 180,E1 29103.465,E2 29103.465} C_VEL
LIN {X 0,Y 759.918,Z 932.862,A -85,B 0,C 180,E1 29102.597,E2 29102.597} C_VEL
LIN {X 0,Y 759.917,Z 957.694,A -85,B 0,C 180,E1 29101.579,E2 29101.579} C_VEL
LIN {X 0,Y 759.912,Z 976.733,A -85,B 0,C 180,E1 29100.698,E2 29100.698} C_VEL
LIN {X 0,Y 759.913,Z 995.417,A -85,B 0,C 180,E1 29099.739,E2 29099.739} C_VEL
LIN {X 0,Y 759.909,Z 1013.698,A -85,B 0,C 180,E1 29098.702,E2 29098.702} C_VEL
LIN {X 0,Y 759.913,Z 1035.188,A -85,B 0,C 180,E1 29097.356,E2 29097.356} C_VEL
LIN {X 0,Y 759.91,Z 1056.55,A -85,B 0,C 180,E1 29095.84,E2 29095.84} C_VEL
LIN {X 0,Y 759.914,Z 1073.31,A -85,B 0,C 180,E1 29094.527,E2 29094.527} C_VEL
LIN {X 0,Y 759.897,Z 1092.039,A -85,B 0,C 180,E1 29092.915,E2 29092.915} C_VEL
LIN {X 0,Y 759.895,Z 1109.491,A -85,B 0,C 180,E1 29091.214,E2 29091.214} C_VEL
LIN {X 0,Y 759.905,Z 1122.956,A -85,B 0,C 180,E1 29089.765,E2 29089.765} C_VEL
LIN {X 0,Y 759.897,Z 1135.73,A -85,B 0,C 180,E1 29088.25,E2 29088.25} C_VEL
LIN {X 0,Y 759.909,Z 1150.03,A -85,B 0,C 180,E1 29086.354,E2 29086.354} C_VEL
LIN {X 0,Y 759.909,Z 1162.193,A -85,B 0,C 180,E1 29084.477,E2 29084.477} C_VEL
LIN {X 0,Y 759.91,Z 1171.058,A -85,B 0,C 180,E1 29082.925,E2 29082.925} C_VEL
LIN {X 0,Y 759.91,Z 1178.784,A -85,B 0,C 180,E1 29081.383,E2 29081.383} C_VEL
LIN {X 0,Y 759.906,Z 1186.43,A -85,B 0,C 180,E1 29079.619,E2 29079.619} C_VEL
LIN {X 0,Y 759.908,Z 1193.594,A -85,B 0,C 180,E1 29077.561,E2 29077.561} C_VEL
LIN {X 0,Y 759.91,Z 1199.108,A -85,B 0,C 180,E1 29075.436,E2 29075.436} C_VEL
LIN {X 0,Y 759.916,Z 1202.585,A -85,B 0,C 180,E1 29073.47,E2 29073.47} C_VEL
LIN {X 0,Y 759.914,Z 1204.58,A -85,B 0,C 180,E1 29071.432,E2 29071.432} C_VEL
LIN {X 0,Y 759.889,Z 1204.849,A -85,B 0,C 180,E1 29069.472,E2 29069.472} C_VEL
LIN {X 0,Y 759.907,Z 1203.906,A -85,B 0,C 180,E1 29067.662,E2 29067.662} C_VEL
LIN {X 0,Y 759.908,Z 1201.053,A -85,B 0,C 180,E1 29065.547,E2 29065.547} C_VEL
LIN {X 0,Y 759.914,Z 1196.566,A -85,B 0,C 180,E1 29063.503,E2 29063.503} C_VEL
LIN {X 0,Y 759.912,Z 1190.628,A -85,B 0,C 180,E1 29061.525,E2 29061.525} C_VEL
LIN {X 0,Y 759.896,Z 1182.679,A -85,B 0,C 180,E1 29059.461,E2 29059.461} C_VEL
LIN {X 0,Y 759.905,Z 1173.109,A -85,B 0,C 180,E1 29057.461,E2 29057.461} C_VEL
LIN {X 0,Y 759.91,Z 1164.053,A -85,B 0,C 180,E1 29055.834,E2 29055.834} C_VEL
LIN {X 0,Y 759.894,Z 1154.208,A -85,B 0,C 180,E1 29054.273,E2 29054.273} C_VEL
LIN {X 0,Y 759.904,Z 1143.662,A -85,B 0,C 180,E1 29052.779,E2 29052.779} C_VEL
LIN {X 0,Y 759.896,Z 1130.456,A -85,B 0,C 180,E1 29051.1,E2 29051.1} C_VEL
LIN {X 0,Y 759.898,Z 1113.388,A -85,B 0,C 180,E1 29049.19,E2 29049.19} C_VEL
LIN {X 0,Y 759.898,Z 1098.821,A -85,B 0,C 180,E1 29047.731,E2 29047.731} C_VEL
LIN {X 0,Y 759.911,Z 1082.646,A -85,B 0,C 180,E1 29046.257,E2 29046.257} C_VEL
LIN {X 0,Y 759.91,Z 1061.264,A -85,B 0,C 180,E1 29044.516,E2 29044.516} C_VEL
LIN {X 0,Y 759.91,Z 1044.038,A -85,B 0,C 180,E1 29043.256,E2 29043.256} C_VEL
LIN {X 0,Y 759.914,Z 1026.229,A -85,B 0,C 180,E1 29042.068,E2 29042.068} C_VEL
LIN {X 0,Y 759.905,Z 1003.437,A -85,B 0,C 180,E1 29040.694,E2 29040.694} C_VEL
LIN {X 0,Y 759.916,Z 981.265,A -85,B 0,C 180,E1 29039.525,E2 29039.525} C_VEL
LIN {X 0,Y 759.912,Z 961.66,A -85,B 0,C 180,E1 29038.597,E2 29038.597} C_VEL
LIN {X 0,Y 759.918,Z 942.461,A -85,B 0,C 180,E1 29037.785,E2 29037.785} C_VEL
LIN {X 0,Y 759.919,Z 923.825,A -85,B 0,C 180,E1 29037.084,E2 29037.084} C_VEL
LIN {X 0,Y 759.909,Z 905.485,A -85,B 0,C 180,E1 29036.473,E2 29036.473} C_VEL
LIN {X 0,Y 759.914,Z 882.794,A -85,B 0,C 180,E1 29035.817,E2 29035.817} C_VEL
LIN {X 0,Y 759.911,Z 855.669,A -85,B 0,C 180,E1 29035.191,E2 29035.191} C_VEL
LIN {X 0,Y 759.909,Z 829.049,A -85,B 0,C 180,E1 29034.736,E2 29034.736} C_VEL
LIN {X 0,Y 759.914,Z 729.625,A -85,B 0,C 180,E1 29033.578,E2 29033.578} C_VEL
LIN {X 0,Y 759.917,Z 507.642,A -85,B 0,C 180,E1 29030.979,E2 29030.979} C_VEL
LIN {X 0,Y 759.905,Z 349.95,A -85,B 0,C 180,E1 29029.06,E2 29029.06} C_VEL
LIN {X 0,Y 759.911,Z 311.066,A -85,B 0,C 180,E1 29026.761,E2 29026.761} C_VEL
LIN {X 0,Y 759.886,Z 309.768,A -85,B 0,C 180,E1 29026.636,E2 29026.636} C_VEL
LIN {X 0,Y 759.825,Z 309.571,A -85,B 0,C 180,E1 29024.069,E2 29024.069} C_VEL
LIN {X 0,Y 759.82,Z 309.576,A -85,B 0,C 180,E1 29021.743,E2 29021.743} C_VEL
LIN {X 0,Y 759.837,Z 309.575,A -85,B 0,C 180,E1 29019.367,E2 29019.367} C_VEL
LIN {X 0,Y 759.907,Z 309.572,A -85,B 0,C 180,E1 29016.491,E2 29016.491} C_VEL
LIN {X 0,Y 759.839,Z 309.573,A -85,B 0,C 180,E1 29013.824,E2 29013.824} C_VEL
LIN {X 0,Y 759.839,Z 309.574,A -85,B 0,C 180,E1 29011.407,E2 29011.407} C_VEL
LIN {X 0,Y 759.913,Z 309.577,A -85,B 0,C 180,E1 29008.703,E2 29008.703} C_VEL
LIN {X 0,Y 759.864,Z 309.57,A -85,B 0,C 180,E1 29005.821,E2 29005.821} C_VEL
LIN {X 0,Y 759.849,Z 309.572,A -85,B 0,C 180,E1 29003.293,E2 29003.293} C_VEL
LIN {X 0,Y 759.916,Z 309.577,A -85,B 0,C 180,E1 29000.568,E2 29000.568} C_VEL
LIN {X 0,Y 759.872,Z 309.568,A -85,B 0,C 180,E1 28997.617,E2 28997.617} C_VEL
LIN {X 0,Y 759.868,Z 309.574,A -85,B 0,C 180,E1 28994.946,E2 28994.946} C_VEL
LIN {X 0,Y 759.908,Z 309.57,A -85,B 0,C 180,E1 28992.141,E2 28992.141} C_VEL
LIN {X 0,Y 759.877,Z 309.568,A -85,B 0,C 180,E1 28989.391,E2 28989.391} C_VEL
LIN {X 0,Y 759.89,Z 309.574,A -85,B 0,C 180,E1 28986.649,E2 28986.649} C_VEL
LIN {X 0,Y 759.912,Z 309.565,A -85,B 0,C 180,E1 28983.697,E2 28983.697} C_VEL
LIN {X 0,Y 759.877,Z 309.57,A -85,B 0,C 180,E1 28980.905,E2 28980.905} C_VEL
LIN {X 0,Y 759.904,Z 309.574,A -85,B 0,C 180,E1 28978.115,E2 28978.115} C_VEL
LIN {X 0,Y 759.888,Z 309.567,A -85,B 0,C 180,E1 28977.089,E2 28977.089} C_VEL
LIN {X 0,Y 758.876,Z 309.703,A -85,B 0,C 180,E1 28976.508,E2 28976.508} C_VEL
LIN {X 0,Y 752.463,Z 310.494,A -85,B 0,C 180,E1 28974.882,E2 28974.882} C_VEL
LIN {X 0,Y 751.96,Z 310.563,A -85,B 0,C 180,E1 28974.459,E2 28974.459} C_VEL
LIN {X 0,Y 751.956,Z 310.556,A -85,B 0,C 180,E1 28971.589,E2 28971.589} C_VEL
LIN {X 0,Y 751.953,Z 310.557,A -85,B 0,C 180,E1 28968.805,E2 28968.805} C_VEL
LIN {X 0,Y 751.963,Z 310.564,A -85,B 0,C 180,E1 28965.995,E2 28965.995} C_VEL
LIN {X 0,Y 751.972,Z 310.552,A -85,B 0,C 180,E1 28963.07,E2 28963.07} C_VEL
LIN {X 0,Y 751.968,Z 310.566,A -85,B 0,C 180,E1 28960.017,E2 28960.017} C_VEL
LIN {X 0,Y 751.951,Z 310.554,A -85,B 0,C 180,E1 28957.145,E2 28957.145} C_VEL
LIN {X 0,Y 751.968,Z 310.562,A -85,B 0,C 180,E1 28954.227,E2 28954.227} C_VEL
LIN {X 0,Y 751.934,Z 310.558,A -85,B 0,C 180,E1 28951.485,E2 28951.485} C_VEL
LIN {X 0,Y 751.971,Z 310.555,A -85,B 0,C 180,E1 28948.674,E2 28948.674} C_VEL
LIN {X 0,Y 751.947,Z 310.565,A -85,B 0,C 180,E1 28945.665,E2 28945.665} C_VEL
LIN {X 0,Y 751.928,Z 310.556,A -85,B 0,C 180,E1 28942.925,E2 28942.925} C_VEL
LIN {X 0,Y 751.973,Z 310.564,A -85,B 0,C 180,E1 28940.041,E2 28940.041} C_VEL
LIN {X 0,Y 751.92,Z 310.564,A -85,B 0,C 180,E1 28937.297,E2 28937.297} C_VEL
LIN {X 0,Y 751.921,Z 310.563,A -85,B 0,C 180,E1 28934.704,E2 28934.704} C_VEL
LIN {X 0,Y 751.965,Z 310.765,A -85,B 0,C 180,E1 28932.467,E2 28932.467} C_VEL
LIN {X 0,Y 753.338,Z 314.722,A -85,B 0,C 180,E1 28932.088,E2 28932.088} C_VEL
LIN {X 0,Y 753.148,Z 355.097,A -85,B 0,C 180,E1 28929.587,E2 28929.587} C_VEL
LIN {X 0,Y 753.053,Z 396.234,A -85,B 0,C 180,E1 28927.13,E2 28927.13} C_VEL
LIN {X 0,Y 753.455,Z 399.754,A -85,B 0,C 180,E1 28927.045,E2 28927.045} C_VEL
LIN {X 0,Y 753.275,Z 643.281,A -85,B 0,C 180,E1 28924.255,E2 28924.255} C_VEL
LIN {X 0,Y 753.107,Z 829.372,A -85,B 0,C 180,E1 28922.162,E2 28922.162} C_VEL
LIN {X 0,Y 753.062,Z 850.051,A -85,B 0,C 180,E1 28921.837,E2 28921.837} C_VEL
LIN {X 0,Y 752.972,Z 876.622,A -85,B 0,C 180,E1 28921.276,E2 28921.276} C_VEL
LIN {X 0,Y 752.903,Z 898.442,A -85,B 0,C 180,E1 28920.684,E2 28920.684} C_VEL
LIN {X 0,Y 752.836,Z 916.981,A -85,B 0,C 180,E1 28920.091,E2 28920.091} C_VEL
LIN {X 0,Y 752.761,Z 936.263,A -85,B 0,C 180,E1 28919.382,E2 28919.382} C_VEL
LIN {X 0,Y 752.665,Z 959.602,A -85,B 0,C 180,E1 28918.398,E2 28918.398} C_VEL
LIN {X 0,Y 752.538,Z 982.435,A -85,B 0,C 180,E1 28917.265,E2 28917.265} C_VEL
LIN {X 0,Y 752.457,Z 1001.858,A -85,B 0,C 180,E1 28916.179,E2 28916.179} C_VEL
LIN {X 0,Y 752.34,Z 1024.424,A -85,B 0,C 180,E1 28914.749,E2 28914.749} C_VEL
LIN {X 0,Y 752.258,Z 1042.035,A -85,B 0,C 180,E1 28913.488,E2 28913.488} C_VEL
LIN {X 0,Y 752.18,Z 1060.948,A -85,B 0,C 180,E1 28911.983,E2 28911.983} C_VEL
LIN {X 0,Y 752.122,Z 1078.364,A -85,B 0,C 180,E1 28910.405,E2 28910.405} C_VEL
LIN {X 0,Y 752.063,Z 1094.59,A -85,B 0,C 180,E1 28908.768,E2 28908.768} C_VEL
LIN {X 0,Y 752.003,Z 1109.379,A -85,B 0,C 180,E1 28907.057,E2 28907.057} C_VEL
LIN {X 0,Y 751.981,Z 1120.759,A -85,B 0,C 180,E1 28905.581,E2 28905.581} C_VEL
LIN {X 0,Y 751.958,Z 1132.62,A -85,B 0,C 180,E1 28903.848,E2 28903.848} C_VEL
LIN {X 0,Y 751.924,Z 1143.504,A -85,B 0,C 180,E1 28901.973,E2 28901.973} C_VEL
LIN {X 0,Y 751.922,Z 1151.236,A -85,B 0,C 180,E1 28900.419,E2 28900.419} C_VEL
LIN {X 0,Y 751.916,Z 1158.109,A -85,B 0,C 180,E1 28898.797,E2 28898.797} C_VEL
LIN {X 0,Y 751.897,Z 1164.757,A -85,B 0,C 180,E1 28896.874,E2 28896.874} C_VEL
LIN {X 0,Y 751.904,Z 1169.571,A -85,B 0,C 180,E1 28894.959,E2 28894.959} C_VEL
LIN {X 0,Y 751.896,Z 1172.447,A -85,B 0,C 180,E1 28893.355,E2 28893.355} C_VEL
LIN {X 0,Y 751.901,Z 1174.368,A -85,B 0,C 180,E1 28891.6,E2 28891.6} C_VEL
LIN {X 0,Y 751.89,Z 1174.885,A -85,B 0,C 180,E1 28889.543,E2 28889.543} C_VEL
LIN {X 0,Y 751.914,Z 1173.977,A -85,B 0,C 180,E1 28887.866,E2 28887.866} C_VEL
LIN {X 0,Y 751.905,Z 1171.903,A -85,B 0,C 180,E1 28886.188,E2 28886.188} C_VEL
LIN {X 0,Y 751.899,Z 1167.636,A -85,B 0,C 180,E1 28884.104,E2 28884.104} C_VEL
LIN {X 0,Y 751.901,Z 1162.796,A -85,B 0,C 180,E1 28882.435,E2 28882.435} C_VEL
LIN {X 0,Y 751.922,Z 1157.247,A -85,B 0,C 180,E1 28880.895,E2 28880.895} C_VEL
LIN {X 0,Y 751.907,Z 1150.226,A -85,B 0,C 180,E1 28879.271,E2 28879.271} C_VEL
LIN {X 0,Y 751.948,Z 1140.185,A -85,B 0,C 180,E1 28877.326,E2 28877.326} C_VEL
LIN {X 0,Y 751.968,Z 1129.572,A -85,B 0,C 180,E1 28875.603,E2 28875.603} C_VEL
LIN {X 0,Y 751.967,Z 1119.1,A -85,B 0,C 180,E1 28874.103,E2 28874.103} C_VEL
LIN {X 0,Y 752.03,Z 1105.334,A -85,B 0,C 180,E1 28872.354,E2 28872.354} C_VEL
LIN {X 0,Y 752.068,Z 1090.022,A -85,B 0,C 180,E1 28870.668,E2 28870.668} C_VEL
LIN {X 0,Y 752.122,Z 1075.275,A -85,B 0,C 180,E1 28869.21,E2 28869.21} C_VEL
LIN {X 0,Y 752.216,Z 1056.145,A -85,B 0,C 180,E1 28867.533,E2 28867.533} C_VEL
LIN {X 0,Y 752.274,Z 1039.205,A -85,B 0,C 180,E1 28866.21,E2 28866.21} C_VEL
LIN {X 0,Y 752.379,Z 1017.584,A -85,B 0,C 180,E1 28864.706,E2 28864.706} C_VEL
LIN {X 0,Y 752.467,Z 999.044,A -85,B 0,C 180,E1 28863.567,E2 28863.567} C_VEL
LIN {X 0,Y 752.548,Z 978.96,A -85,B 0,C 180,E1 28862.46,E2 28862.46} C_VEL
LIN {X 0,Y 752.683,Z 954.741,A -85,B 0,C 180,E1 28861.3,E2 28861.3} C_VEL
LIN {X 0,Y 752.767,Z 934.585,A -85,B 0,C 180,E1 28860.462,E2 28860.462} C_VEL
LIN {X 0,Y 752.837,Z 914.381,A -85,B 0,C 180,E1 28859.729,E2 28859.729} C_VEL
LIN {X 0,Y 752.954,Z 889.05,A -85,B 0,C 180,E1 28858.954,E2 28858.954} C_VEL
LIN {X 0,Y 753.014,Z 866.314,A -85,B 0,C 180,E1 28858.4,E2 28858.4} C_VEL
LIN {X 0,Y 753.07,Z 846.438,A -85,B 0,C 180,E1 28858.011,E2 28858.011} C_VEL
LIN {X 0,Y 753.111,Z 826.948,A -85,B 0,C 180,E1 28857.716,E2 28857.716} C_VEL
LIN {X 0,Y 753.326,Z 569.295,A -85,B 0,C 180,E1 28854.818,E2 28854.818} C_VEL
LIN {X 0,Y 753.355,Z 398.015,A -85,B 0,C 180,E1 28852.839,E2 28852.839} C_VEL
LIN {X 0,Y 753.019,Z 395.386,A -85,B 0,C 180,E1 28852.736,E2 28852.736} C_VEL
LIN {X 0,Y 753.16,Z 353.343,A -85,B 0,C 180,E1 28850.217,E2 28850.217} C_VEL
LIN {X 0,Y 753.332,Z 314.148,A -85,B 0,C 180,E1 28847.785,E2 28847.785} C_VEL
LIN {X 0,Y 751.941,Z 310.704,A -85,B 0,C 180,E1 28847.426,E2 28847.426} C_VEL
LIN {X 0,Y 751.901,Z 310.566,A -85,B 0,C 180,E1 28844.921,E2 28844.921} C_VEL
LIN {X 0,Y 751.936,Z 310.566,A -85,B 0,C 180,E1 28842.391,E2 28842.391} C_VEL
LIN {X 0,Y 751.937,Z 310.559,A -85,B 0,C 180,E1 28839.294,E2 28839.294} C_VEL
LIN {X 0,Y 751.915,Z 310.56,A -85,B 0,C 180,E1 28836.693,E2 28836.693} C_VEL
LIN {X 0,Y 751.976,Z 310.562,A -85,B 0,C 180,E1 28833.931,E2 28833.931} C_VEL
LIN {X 0,Y 751.941,Z 310.557,A -85,B 0,C 180,E1 28831.061,E2 28831.061} C_VEL
LIN {X 0,Y 751.936,Z 310.56,A -85,B 0,C 180,E1 28828.324,E2 28828.324} C_VEL
LIN {X 0,Y 751.968,Z 310.557,A -85,B 0,C 180,E1 28825.465,E2 28825.465} C_VEL
LIN {X 0,Y 751.937,Z 310.557,A -85,B 0,C 180,E1 28822.656,E2 28822.656} C_VEL
LIN {X 0,Y 751.977,Z 310.563,A -85,B 0,C 180,E1 28819.82,E2 28819.82} C_VEL
LIN {X 0,Y 751.961,Z 310.554,A -85,B 0,C 180,E1 28816.789,E2 28816.789} C_VEL
LIN {X 0,Y 751.972,Z 310.566,A -85,B 0,C 180,E1 28813.848,E2 28813.848} C_VEL
LIN {X 0,Y 751.975,Z 310.552,A -85,B 0,C 180,E1 28810.806,E2 28810.806} C_VEL
LIN {X 0,Y 751.972,Z 310.565,A -85,B 0,C 180,E1 28807.795,E2 28807.795} C_VEL
LIN {X 0,Y 751.962,Z 310.554,A -85,B 0,C 180,E1 28804.805,E2 28804.805} C_VEL
LIN {X 0,Y 751.961,Z 310.562,A -85,B 0,C 180,E1 28801.905,E2 28801.905} C_VEL
LIN {X 0,Y 751.944,Z 310.56,A -85,B 0,C 180,E1 28799.162,E2 28799.162} C_VEL
LIN {X 0,Y 751.975,Z 310.554,A -85,B 0,C 180,E1 28796.341,E2 28796.341} C_VEL
LIN {X 0,Y 751.956,Z 310.563,A -85,B 0,C 180,E1 28793.355,E2 28793.355} C_VEL
LIN {X 0,Y 751.947,Z 310.556,A -85,B 0,C 180,E1 28790.509,E2 28790.509} C_VEL
LIN {X 0,Y 751.976,Z 310.562,A -85,B 0,C 180,E1 28787.56,E2 28787.56} C_VEL
LIN {X 0,Y 751.925,Z 310.561,A -85,B 0,C 180,E1 28784.813,E2 28784.813} C_VEL
LIN {X 0,Y 751.963,Z 310.553,A -85,B 0,C 180,E1 28782.112,E2 28782.112} C_VEL
LIN {X 0,Y 751.942,Z 310.564,A -85,B 0,C 180,E1 28779.122,E2 28779.122} C_VEL
LIN {X 0,Y 751.913,Z 310.558,A -85,B 0,C 180,E1 28776.488,E2 28776.488} C_VEL
LIN {X 0,Y 751.975,Z 310.559,A -85,B 0,C 180,E1 28773.718,E2 28773.718} C_VEL
LIN {X 0,Y 751.921,Z 310.564,A -85,B 0,C 180,E1 28770.876,E2 28770.876} C_VEL
LIN {X 0,Y 751.899,Z 310.561,A -85,B 0,C 180,E1 28768.402,E2 28768.402} C_VEL
LIN {X 0,Y 751.929,Z 310.56,A -85,B 0,C 180,E1 28765.864,E2 28765.864} C_VEL
LIN {X 0,Y 751.915,Z 310.566,A -85,B 0,C 180,E1 28762.8,E2 28762.8} C_VEL
LIN {X 0,Y 751.885,Z 310.562,A -85,B 0,C 180,E1 28760.333,E2 28760.333} C_VEL
LIN {X 0,Y 751.888,Z 310.565,A -85,B 0,C 180,E1 28758.017,E2 28758.017} C_VEL
LIN {X 0,Y 751.976,Z 310.527,A -85,B 0,C 180,E1 28755.192,E2 28755.192} C_VEL
LIN {X 0,Y 751.903,Z 310.697,A -85,B 0,C 180,E1 28753.883,E2 28753.883} C_VEL
LIN {X 0,Y 753.174,Z 313.966,A -85,B 0,C 180,E1 28753.543,E2 28753.543} C_VEL
LIN {X 0,Y 753.469,Z 315.559,A -85,B 0,C 180,E1 28753.425,E2 28753.425} C_VEL
LIN {X 0,Y 753.472,Z 350.651,A -85,B 0,C 180,E1 28751.346,E2 28751.346} C_VEL
LIN {X 0,Y 753.836,Z 353.985,A -85,B 0,C 180,E1 28751.277,E2 28751.277} C_VEL
LIN {X 0,Y 753.625,Z 567.13,A -85,B 0,C 180,E1 28748.694,E2 28748.694} C_VEL
LIN {X 0,Y 753.408,Z 793.203,A -85,B 0,C 180,E1 28746.051,E2 28746.051} C_VEL
LIN {X 0,Y 753.349,Z 832.599,A -85,B 0,C 180,E1 28745.565,E2 28745.565} C_VEL
LIN {X 0,Y 753.271,Z 858.76,A -85,B 0,C 180,E1 28745.095,E2 28745.095} C_VEL
LIN {X 0,Y 753.187,Z 885.204,A -85,B 0,C 180,E1 28744.468,E2 28744.468} C_VEL
LIN {X 0,Y 753.089,Z 911.426,A -85,B 0,C 180,E1 28743.686,E2 28743.686} C_VEL
LIN {X 0,Y 752.955,Z 937.233,A -85,B 0,C 180,E1 28742.761,E2 28742.761} C_VEL
LIN {X 0,Y 752.856,Z 958.691,A -85,B 0,C 180,E1 28741.865,E2 28741.865} C_VEL
LIN {X 0,Y 752.759,Z 977.627,A -85,B 0,C 180,E1 28740.978,E2 28740.978} C_VEL
LIN {X 0,Y 752.665,Z 996.704,A -85,B 0,C 180,E1 28739.984,E2 28739.984} C_VEL
LIN {X 0,Y 752.56,Z 1016.612,A -85,B 0,C 180,E1 28738.835,E2 28738.835} C_VEL
LIN {X 0,Y 752.413,Z 1040.415,A -85,B 0,C 180,E1 28737.288,E2 28737.288} C_VEL
LIN {X 0,Y 752.343,Z 1058.5,A -85,B 0,C 180,E1 28735.97,E2 28735.97} C_VEL
LIN {X 0,Y 752.262,Z 1076.357,A -85,B 0,C 180,E1 28734.542,E2 28734.542} C_VEL
LIN {X 0,Y 752.17,Z 1096.265,A -85,B 0,C 180,E1 28732.757,E2 28732.757} C_VEL
LIN {X 0,Y 752.096,Z 1111.282,A -85,B 0,C 180,E1 28731.257,E2 28731.257} C_VEL
LIN {X 0,Y 752.063,Z 1125.174,A -85,B 0,C 180,E1 28729.727,E2 28729.727} C_VEL
LIN {X 0,Y 752.008,Z 1141.337,A -85,B 0,C 180,E1 28727.727,E2 28727.727} C_VEL
LIN {X 0,Y 751.956,Z 1153.167,A -85,B 0,C 180,E1 28726.056,E2 28726.056} C_VEL
LIN {X 0,Y 751.954,Z 1163.126,A -85,B 0,C 180,E1 28724.476,E2 28724.476} C_VEL
LIN {X 0,Y 751.94,Z 1171.88,A -85,B 0,C 180,E1 28722.908,E2 28722.908} C_VEL
LIN {X 0,Y 751.93,Z 1179.5,A -85,B 0,C 180,E1 28721.35,E2 28721.35} C_VEL
LIN {X 0,Y 751.916,Z 1187.31,A -85,B 0,C 180,E1 28719.491,E2 28719.491} C_VEL
LIN {X 0,Y 751.911,Z 1194.033,A -85,B 0,C 180,E1 28717.488,E2 28717.488} C_VEL
LIN {X 0,Y 751.911,Z 1199.28,A -85,B 0,C 180,E1 28715.417,E2 28715.417} C_VEL
LIN {X 0,Y 751.914,Z 1202.789,A -85,B 0,C 180,E1 28713.354,E2 28713.354} C_VEL
LIN {X 0,Y 751.915,Z 1204.603,A -85,B 0,C 180,E1 28711.371,E2 28711.371} C_VEL
LIN {X 0,Y 751.889,Z 1204.849,A -85,B 0,C 180,E1 28709.466,E2 28709.466} C_VEL
LIN {X 0,Y 751.907,Z 1203.906,A -85,B 0,C 180,E1 28707.637,E2 28707.637} C_VEL
LIN {X 0,Y 751.907,Z 1201.053,A -85,B 0,C 180,E1 28705.5,E2 28705.5} C_VEL
LIN {X 0,Y 751.912,Z 1196.565,A -85,B 0,C 180,E1 28703.433,E2 28703.433} C_VEL
LIN {X 0,Y 751.92,Z 1190.628,A -85,B 0,C 180,E1 28701.435,E2 28701.435} C_VEL
LIN {X 0,Y 751.905,Z 1182.636,A -85,B 0,C 180,E1 28699.338,E2 28699.338} C_VEL
LIN {X 0,Y 751.935,Z 1173.11,A -85,B 0,C 180,E1 28697.326,E2 28697.326} C_VEL
LIN {X 0,Y 751.955,Z 1164.055,A -85,B 0,C 180,E1 28695.681,E2 28695.681} C_VEL
LIN {X 0,Y 751.954,Z 1154.21,A -85,B 0,C 180,E1 28694.102,E2 28694.102} C_VEL
LIN {X 0,Y 752.006,Z 1143.082,A -85,B 0,C 180,E1 28692.513,E2 28692.513} C_VEL
LIN {X 0,Y 752.065,Z 1127.927,A -85,B 0,C 180,E1 28690.587,E2 28690.587} C_VEL
LIN {X 0,Y 752.088,Z 1112.61,A -85,B 0,C 180,E1 28688.882,E2 28688.882} C_VEL
LIN {X 0,Y 752.167,Z 1097.969,A -85,B 0,C 180,E1 28687.407,E2 28687.407} C_VEL
LIN {X 0,Y 752.232,Z 1079.851,A -85,B 0,C 180,E1 28685.749,E2 28685.749} C_VEL
LIN {X 0,Y 752.346,Z 1060.156,A -85,B 0,C 180,E1 28684.156,E2 28684.156} C_VEL
LIN {X 0,Y 752.409,Z 1042.829,A -85,B 0,C 180,E1 28682.883,E2 28682.883} C_VEL
LIN {X 0,Y 752.521,Z 1022.257,A -85,B 0,C 180,E1 28681.51,E2 28681.51} C_VEL
LIN {X 0,Y 752.657,Z 998.623,A -85,B 0,C 180,E1 28680.121,E2 28680.121} C_VEL
LIN {X 0,Y 752.754,Z 979.256,A -85,B 0,C 180,E1 28679.103,E2 28679.103} C_VEL
LIN {X 0,Y 752.85,Z 960.434,A -85,B 0,C 180,E1 28678.213,E2 28678.213} C_VEL
LIN {X 0,Y 752.949,Z 940.579,A -85,B 0,C 180,E1 28677.374,E2 28677.374} C_VEL
LIN {X 0,Y 753.037,Z 920.015,A -85,B 0,C 180,E1 28676.607,E2 28676.607} C_VEL
LIN {X 0,Y 753.158,Z 894.913,A -85,B 0,C 180,E1 28675.802,E2 28675.802} C_VEL
LIN {X 0,Y 753.243,Z 867.527,A -85,B 0,C 180,E1 28675.096,E2 28675.096} C_VEL
LIN {X 0,Y 753.329,Z 841.967,A -85,B 0,C 180,E1 28674.587,E2 28674.587} C_VEL
LIN {X 0,Y 753.38,Z 814.848,A -85,B 0,C 180,E1 28674.197,E2 28674.197} C_VEL
LIN {X 0,Y 753.596,Z 589.203,A -85,B 0,C 180,E1 28671.568,E2 28671.568} C_VEL
LIN {X 0,Y 753.785,Z 382.551,A -85,B 0,C 180,E1 28669.073,E2 28669.073} C_VEL
LIN {X 0,Y 753.651,Z 351.479,A -85,B 0,C 180,E1 28668.679,E2 28668.679} C_VEL
LIN {X 0,Y 753.347,Z 349.135,A -85,B 0,C 180,E1 28668.582,E2 28668.582} C_VEL
LIN {X 0,Y 753.399,Z 314.309,A -85,B 0,C 180,E1 28666.494,E2 28666.494} C_VEL
LIN {X 0,Y 751.918,Z 310.794,A -85,B 0,C 180,E1 28666.133,E2 28666.133} C_VEL
LIN {X 0,Y 751.88,Z 310.553,A -85,B 0,C 180,E1 28663.962,E2 28663.962} C_VEL
LIN {X 0,Y 751.883,Z 310.566,A -85,B 0,C 180,E1 28661.637,E2 28661.637} C_VEL
LIN {X 0,Y 751.931,Z 310.564,A -85,B 0,C 180,E1 28659.073,E2 28659.073} C_VEL
LIN {X 0,Y 751.915,Z 310.561,A -85,B 0,C 180,E1 28656.093,E2 28656.093} C_VEL
LIN {X 0,Y 751.896,Z 310.563,A -85,B 0,C 180,E1 28653.648,E2 28653.648} C_VEL
LIN {X 0,Y 751.916,Z 310.564,A -85,B 0,C 180,E1 28651.151,E2 28651.151} C_VEL
LIN {X 0,Y 751.96,Z 310.556,A -85,B 0,C 180,E1 28648.167,E2 28648.167} C_VEL
LIN {X 0,Y 751.908,Z 310.561,A -85,B 0,C 180,E1 28645.522,E2 28645.522} C_VEL
LIN {X 0,Y 751.934,Z 310.562,A -85,B 0,C 180,E1 28642.931,E2 28642.931} C_VEL
LIN {X 0,Y 751.957,Z 310.556,A -85,B 0,C 180,E1 28639.902,E2 28639.902} C_VEL
LIN {X 0,Y 751.919,Z 310.558,A -85,B 0,C 180,E1 28637.25,E2 28637.25} C_VEL
LIN {X 0,Y 751.979,Z 310.565,A -85,B 0,C 180,E1 28634.476,E2 28634.476} C_VEL
LIN {X 0,Y 751.942,Z 310.554,A -85,B 0,C 180,E1 28631.506,E2 28631.506} C_VEL
LIN {X 0,Y 751.947,Z 310.564,A -85,B 0,C 180,E1 28628.719,E2 28628.719} C_VEL
LIN {X 0,Y 751.973,Z 310.552,A -85,B 0,C 180,E1 28625.723,E2 28625.723} C_VEL
LIN {X 0,Y 751.938,Z 310.561,A -85,B 0,C 180,E1 28622.896,E2 28622.896} C_VEL
LIN {X 0,Y 751.967,Z 310.56,A -85,B 0,C 180,E1 28620.152,E2 28620.152} C_VEL
LIN {X 0,Y 751.962,Z 310.554,A -85,B 0,C 180,E1 28617.256,E2 28617.256} C_VEL
LIN {X 0,Y 751.96,Z 310.563,A -85,B 0,C 180,E1 28614.459,E2 28614.459} C_VEL
LIN {X 0,Y 751.004,Z 310.692,A -85,B 0,C 180,E1 28613.872,E2 28613.872} C_VEL
LIN {X 0,Y 744.555,Z 311.489,A -85,B 0,C 180,E1 28612.229,E2 28612.229} C_VEL
LIN {X 0,Y 744.015,Z 311.548,A -85,B 0,C 180,E1 28611.802,E2 28611.802} C_VEL
LIN {X 0,Y 744.024,Z 311.543,A -85,B 0,C 180,E1 28608.999,E2 28608.999} C_VEL
LIN {X 0,Y 744.031,Z 311.554,A -85,B 0,C 180,E1 28606.081,E2 28606.081} C_VEL
LIN {X 0,Y 744.033,Z 311.541,A -85,B 0,C 180,E1 28603.045,E2 28603.045} C_VEL
LIN {X 0,Y 744.031,Z 311.554,A -85,B 0,C 180,E1 28600.041,E2 28600.041} C_VEL
LIN {X 0,Y 744.012,Z 311.543,A -85,B 0,C 180,E1 28597.145,E2 28597.145} C_VEL
LIN {X 0,Y 744.031,Z 311.551,A -85,B 0,C 180,E1 28594.188,E2 28594.188} C_VEL
LIN {X 0,Y 743.993,Z 311.545,A -85,B 0,C 180,E1 28591.416,E2 28591.416} C_VEL
LIN {X 0,Y 744.034,Z 311.544,A -85,B 0,C 180,E1 28588.662,E2 28588.662} C_VEL
LIN {X 0,Y 744.006,Z 311.554,A -85,B 0,C 180,E1 28585.636,E2 28585.636} C_VEL
LIN {X 0,Y 743.993,Z 311.544,A -85,B 0,C 180,E1 28582.884,E2 28582.884} C_VEL
LIN {X 0,Y 744.038,Z 311.552,A -85,B 0,C 180,E1 28579.93,E2 28579.93} C_VEL
LIN {X 0,Y 743.976,Z 311.553,A -85,B 0,C 180,E1 28577.152,E2 28577.152} C_VEL
LIN {X 0,Y 743.997,Z 311.553,A -85,B 0,C 180,E1 28574.55,E2 28574.55} C_VEL
LIN {X 0,Y 743.988,Z 311.689,A -85,B 0,C 180,E1 28572.984,E2 28572.984} C_VEL
LIN {X 0,Y 745.112,Z 314.757,A -85,B 0,C 180,E1 28572.66,E2 28572.66} C_VEL
LIN {X 0,Y 746.769,Z 318.73,A -85,B 0,C 180,E1 28572.288,E2 28572.288} C_VEL
LIN {X 0,Y 746.419,Z 359.513,A -85,B 0,C 180,E1 28569.743,E2 28569.743} C_VEL
LIN {X 0,Y 746.237,Z 396.559,A -85,B 0,C 180,E1 28567.512,E2 28567.512} C_VEL
LIN {X 0,Y 747.059,Z 401.329,A -85,B 0,C 180,E1 28567.398,E2 28567.398} C_VEL
LIN {X 0,Y 746.653,Z 645.81,A -85,B 0,C 180,E1 28564.573,E2 28564.573} C_VEL
LIN {X 0,Y 746.324,Z 829.416,A -85,B 0,C 180,E1 28562.49,E2 28562.49} C_VEL
LIN {X 0,Y 746.234,Z 850.796,A -85,B 0,C 180,E1 28562.151,E2 28562.151} C_VEL
LIN {X 0,Y 746.05,Z 878.158,A -85,B 0,C 180,E1 28561.56,E2 28561.56} C_VEL
LIN {X 0,Y 745.913,Z 899.198,A -85,B 0,C 180,E1 28560.98,E2 28560.98} C_VEL
LIN {X 0,Y 745.773,Z 918.272,A -85,B 0,C 180,E1 28560.362,E2 28560.362} C_VEL
LIN {X 0,Y 745.607,Z 940.467,A -85,B 0,C 180,E1 28559.527,E2 28559.527} C_VEL
LIN {X 0,Y 745.347,Z 964.987,A -85,B 0,C 180,E1 28558.44,E2 28558.44} C_VEL
LIN {X 0,Y 745.173,Z 984.502,A -85,B 0,C 180,E1 28557.446,E2 28557.446} C_VEL
LIN {X 0,Y 744.996,Z 1006.221,A -85,B 0,C 180,E1 28556.204,E2 28556.204} C_VEL
LIN {X 0,Y 744.763,Z 1027.148,A -85,B 0,C 180,E1 28554.827,E2 28554.827} C_VEL
LIN {X 0,Y 744.616,Z 1045.432,A -85,B 0,C 180,E1 28553.486,E2 28553.486} C_VEL
LIN {X 0,Y 744.431,Z 1064.303,A -85,B 0,C 180,E1 28551.925,E2 28551.925} C_VEL
LIN {X 0,Y 744.334,Z 1079.447,A -85,B 0,C 180,E1 28550.525,E2 28550.525} C_VEL
LIN {X 0,Y 744.206,Z 1096.045,A -85,B 0,C 180,E1 28548.811,E2 28548.811} C_VEL
LIN {X 0,Y 744.109,Z 1109.929,A -85,B 0,C 180,E1 28547.175,E2 28547.175} C_VEL
LIN {X 0,Y 744.052,Z 1121.345,A -85,B 0,C 180,E1 28545.671,E2 28545.671} C_VEL
LIN {X 0,Y 743.999,Z 1133.622,A -85,B 0,C 180,E1 28543.841,E2 28543.841} C_VEL
LIN {X 0,Y 743.95,Z 1143.917,A -85,B 0,C 180,E1 28542.024,E2 28542.024} C_VEL
LIN {X 0,Y 743.935,Z 1151.595,A -85,B 0,C 180,E1 28540.454,E2 28540.454} C_VEL
LIN {X 0,Y 743.922,Z 1158.721,A -85,B 0,C 180,E1 28538.736,E2 28538.736} C_VEL
LIN {X 0,Y 743.899,Z 1165.604,A -85,B 0,C 180,E1 28536.631,E2 28536.631} C_VEL
LIN {X 0,Y 743.903,Z 1169.732,A -85,B 0,C 180,E1 28534.935,E2 28534.935} C_VEL
LIN {X 0,Y 743.899,Z 1172.56,A -85,B 0,C 180,E1 28533.313,E2 28533.313} C_VEL
LIN {X 0,Y 743.908,Z 1174.569,A -85,B 0,C 180,E1 28531.386,E2 28531.386} C_VEL
LIN {X 0,Y 743.889,Z 1174.863,A -85,B 0,C 180,E1 28529.461,E2 28529.461} C_VEL
LIN {X 0,Y 743.914,Z 1173.977,A -85,B 0,C 180,E1 28527.843,E2 28527.843} C_VEL
LIN {X 0,Y 743.909,Z 1171.903,A -85,B 0,C 180,E1 28526.147,E2 28526.147} C_VEL
LIN {X 0,Y 743.903,Z 1167.686,A -85,B 0,C 180,E1 28524.06,E2 28524.06} C_VEL
LIN {X 0,Y 743.909,Z 1162.795,A -85,B 0,C 180,E1 28522.353,E2 28522.353} C_VEL
LIN {X 0,Y 743.932,Z 1157.245,A -85,B 0,C 180,E1 28520.797,E2 28520.797} C_VEL
LIN {X 0,Y 743.922,Z 1150.225,A -85,B 0,C 180,E1 28519.154,E2 28519.154} C_VEL
LIN {X 0,Y 743.986,Z 1140.183,A -85,B 0,C 180,E1 28517.188,E2 28517.188} C_VEL
LIN {X 0,Y 744.02,Z 1129.57,A -85,B 0,C 180,E1 28515.445,E2 28515.445} C_VEL
LIN {X 0,Y 744.046,Z 1119.011,A -85,B 0,C 180,E1 28513.917,E2 28513.917} C_VEL
LIN {X 0,Y 744.147,Z 1105.328,A -85,B 0,C 180,E1 28512.161,E2 28512.161} C_VEL
LIN {X 0,Y 744.246,Z 1090.019,A -85,B 0,C 180,E1 28510.457,E2 28510.457} C_VEL
LIN {X 0,Y 744.339,Z 1075.27,A -85,B 0,C 180,E1 28508.982,E2 28508.982} C_VEL
LIN {X 0,Y 744.523,Z 1056.475,A -85,B 0,C 180,E1 28507.315,E2 28507.315} C_VEL
LIN {X 0,Y 744.646,Z 1039.752,A -85,B 0,C 180,E1 28505.993,E2 28505.993} C_VEL
LIN {X 0,Y 744.862,Z 1018.902,A -85,B 0,C 180,E1 28504.518,E2 28504.518} C_VEL
LIN {X 0,Y 745.037,Z 999.037,A -85,B 0,C 180,E1 28503.283,E2 28503.283} C_VEL
LIN {X 0,Y 745.232,Z 978.148,A -85,B 0,C 180,E1 28502.123,E2 28502.123} C_VEL
LIN {X 0,Y 745.472,Z 954.553,A -85,B 0,C 180,E1 28500.988,E2 28500.988} C_VEL
LIN {X 0,Y 745.632,Z 934.927,A -85,B 0,C 180,E1 28500.165,E2 28500.165} C_VEL
LIN {X 0,Y 745.786,Z 914.041,A -85,B 0,C 180,E1 28499.401,E2 28499.401} C_VEL
LIN {X 0,Y 746.024,Z 887.551,A -85,B 0,C 180,E1 28498.595,E2 28498.595} C_VEL
LIN {X 0,Y 746.143,Z 865.642,A -85,B 0,C 180,E1 28498.06,E2 28498.06} C_VEL
LIN {X 0,Y 746.249,Z 845.598,A -85,B 0,C 180,E1 28497.669,E2 28497.669} C_VEL
LIN {X 0,Y 746.333,Z 825.193,A -85,B 0,C 180,E1 28497.364,E2 28497.364} C_VEL
LIN {X 0,Y 746.773,Z 571.774,A -85,B 0,C 180,E1 28494.492,E2 28494.492} C_VEL
LIN {X 0,Y 746.992,Z 399.975,A -85,B 0,C 180,E1 28492.492,E2 28492.492} C_VEL
LIN {X 0,Y 746.202,Z 395.9,A -85,B 0,C 180,E1 28492.366,E2 28492.366} C_VEL
LIN {X 0,Y 746.499,Z 352.524,A -85,B 0,C 180,E1 28489.739,E2 28489.739} C_VEL
LIN {X 0,Y 746.765,Z 318.368,A -85,B 0,C 180,E1 28487.599,E2 28487.599} C_VEL
LIN {X 0,Y 744.026,Z 311.982,A -85,B 0,C 180,E1 28486.977,E2 28486.977} C_VEL
LIN {X 0,Y 743.973,Z 311.539,A -85,B 0,C 180,E1 28486.625,E2 28486.625} C_VEL
LIN {X 0,Y 744.037,Z 311.549,A -85,B 0,C 180,E1 28483.698,E2 28483.698} C_VEL
LIN {X 0,Y 743.97,Z 311.546,A -85,B 0,C 180,E1 28480.948,E2 28480.948} C_VEL
LIN {X 0,Y 744.006,Z 311.556,A -85,B 0,C 180,E1 28478.284,E2 28478.284} C_VEL
LIN {X 0,Y 744.004,Z 311.547,A -85,B 0,C 180,E1 28475.205,E2 28475.205} C_VEL
LIN {X 0,Y 743.985,Z 311.548,A -85,B 0,C 180,E1 28472.52,E2 28472.52} C_VEL
LIN {X 0,Y 744.031,Z 311.546,A -85,B 0,C 180,E1 28469.729,E2 28469.729} C_VEL
LIN {X 0,Y 743.998,Z 311.547,A -85,B 0,C 180,E1 28466.844,E2 28466.844} C_VEL
LIN {X 0,Y 744.023,Z 311.551,A -85,B 0,C 180,E1 28464.029,E2 28464.029} C_VEL
LIN {X 0,Y 744.023,Z 311.544,A -85,B 0,C 180,E1 28460.934,E2 28460.934} C_VEL
LIN {X 0,Y 744.02,Z 311.549,A -85,B 0,C 180,E1 28458.005,E2 28458.005} C_VEL
LIN {X 0,Y 744.032,Z 311.543,A -85,B 0,C 180,E1 28455.033,E2 28455.033} C_VEL
LIN {X 0,Y 744.009,Z 311.544,A -85,B 0,C 180,E1 28452.181,E2 28452.181} C_VEL
LIN {X 0,Y 744.016,Z 311.55,A -85,B 0,C 180,E1 28449.359,E2 28449.359} C_VEL
LIN {X 0,Y 744.023,Z 311.538,A -85,B 0,C 180,E1 28446.482,E2 28446.482} C_VEL
LIN {X 0,Y 744.029,Z 311.554,A -85,B 0,C 180,E1 28443.544,E2 28443.544} C_VEL
LIN {X 0,Y 744.035,Z 311.537,A -85,B 0,C 180,E1 28440.539,E2 28440.539} C_VEL
LIN {X 0,Y 744.025,Z 311.554,A -85,B 0,C 180,E1 28437.458,E2 28437.458} C_VEL
LIN {X 0,Y 744.02,Z 311.54,A -85,B 0,C 180,E1 28434.525,E2 28434.525} C_VEL
LIN {X 0,Y 744.033,Z 311.555,A -85,B 0,C 180,E1 28431.499,E2 28431.499} C_VEL
LIN {X 0,Y 743.993,Z 311.544,A -85,B 0,C 180,E1 28428.684,E2 28428.684} C_VEL
LIN {X 0,Y 744.031,Z 311.546,A -85,B 0,C 180,E1 28425.843,E2 28425.843} C_VEL
LIN {X 0,Y 743.993,Z 311.548,A -85,B 0,C 180,E1 28423.044,E2 28423.044} C_VEL
LIN {X 0,Y 743.991,Z 311.547,A -85,B 0,C 180,E1 28420.367,E2 28420.367} C_VEL
LIN {X 0,Y 744.035,Z 311.55,A -85,B 0,C 180,E1 28417.397,E2 28417.397} C_VEL
LIN {X 0,Y 743.974,Z 311.552,A -85,B 0,C 180,E1 28414.698,E2 28414.698} C_VEL
LIN {X 0,Y 743.986,Z 311.545,A -85,B 0,C 180,E1 28412.115,E2 28412.115} C_VEL
LIN {X 0,Y 744.012,Z 311.553,A -85,B 0,C 180,E1 28409.111,E2 28409.111} C_VEL
LIN {X 0,Y 743.958,Z 311.552,A -85,B 0,C 180,E1 28406.469,E2 28406.469} C_VEL
LIN {X 0,Y 743.969,Z 311.55,A -85,B 0,C 180,E1 28404.005,E2 28404.005} C_VEL
LIN {X 0,Y 744.02,Z 311.552,A -85,B 0,C 180,E1 28401.087,E2 28401.087} C_VEL
LIN {X 0,Y 743.946,Z 311.556,A -85,B 0,C 180,E1 28398.398,E2 28398.398} C_VEL
LIN {X 0,Y 743.94,Z 311.536,A -85,B 0,C 180,E1 28396.087,E2 28396.087} C_VEL
LIN {X 0,Y 743.967,Z 311.715,A -85,B 0,C 180,E1 28394.403,E2 28394.403} C_VEL
LIN {X 0,Y 745.42,Z 315.295,A -85,B 0,C 180,E1 28394.029,E2 28394.029} C_VEL
LIN {X 0,Y 747.039,Z 318.991,A -85,B 0,C 180,E1 28393.681,E2 28393.681} C_VEL
LIN {X 0,Y 746.944,Z 350.712,A -85,B 0,C 180,E1 28391.787,E2 28391.787} C_VEL
LIN {X 0,Y 747.805,Z 355.244,A -85,B 0,C 180,E1 28391.668,E2 28391.668} C_VEL
LIN {X 0,Y 747.366,Z 568.472,A -85,B 0,C 180,E1 28389.063,E2 28389.063} C_VEL
LIN {X 0,Y 746.928,Z 794.233,A -85,B 0,C 180,E1 28386.401,E2 28386.401} C_VEL
LIN {X 0,Y 746.815,Z 833.231,A -85,B 0,C 180,E1 28385.915,E2 28385.915} C_VEL
LIN {X 0,Y 746.66,Z 859.609,A -85,B 0,C 180,E1 28385.433,E2 28385.433} C_VEL
LIN {X 0,Y 746.489,Z 885.764,A -85,B 0,C 180,E1 28384.806,E2 28384.806} C_VEL
LIN {X 0,Y 746.286,Z 913.615,A -85,B 0,C 180,E1 28383.966,E2 28383.966} C_VEL
LIN {X 0,Y 746.007,Z 939.473,A -85,B 0,C 180,E1 28383.013,E2 28383.013} C_VEL
LIN {X 0,Y 745.814,Z 959.688,A -85,B 0,C 180,E1 28382.157,E2 28382.157} C_VEL
LIN {X 0,Y 745.617,Z 979.499,A -85,B 0,C 180,E1 28381.213,E2 28381.213} C_VEL
LIN {X 0,Y 745.41,Z 1001.041,A -85,B 0,C 180,E1 28380.066,E2 28380.066} C_VEL
LIN {X 0,Y 745.121,Z 1024.914,A -85,B 0,C 180,E1 28378.624,E2 28378.624} C_VEL
LIN {X 0,Y 744.926,Z 1043.44,A -85,B 0,C 180,E1 28377.369,E2 28377.369} C_VEL
LIN {X 0,Y 744.78,Z 1061.269,A -85,B 0,C 180,E1 28376.04,E2 28376.04} C_VEL
LIN {X 0,Y 744.534,Z 1082.651,A -85,B 0,C 180,E1 28374.264,E2 28374.264} C_VEL
LIN {X 0,Y 744.424,Z 1098.827,A -85,B 0,C 180,E1 28372.757,E2 28372.757} C_VEL
LIN {X 0,Y 744.287,Z 1114.955,A -85,B 0,C 180,E1 28371.102,E2 28371.102} C_VEL
LIN {X 0,Y 744.155,Z 1131.865,A -85,B 0,C 180,E1 28369.138,E2 28369.138} C_VEL
LIN {X 0,Y 744.097,Z 1144.25,A -85,B 0,C 180,E1 28367.517,E2 28367.517} C_VEL
LIN {X 0,Y 744.02,Z 1154.736,A -85,B 0,C 180,E1 28365.991,E2 28365.991} C_VEL
LIN {X 0,Y 743.999,Z 1164.524,A -85,B 0,C 180,E1 28364.396,E2 28364.396} C_VEL
LIN {X 0,Y 743.961,Z 1174.755,A -85,B 0,C 180,E1 28362.496,E2 28362.496} C_VEL
LIN {X 0,Y 743.933,Z 1184.913,A -85,B 0,C 180,E1 28360.219,E2 28360.219} C_VEL
LIN {X 0,Y 743.923,Z 1191.892,A -85,B 0,C 180,E1 28358.268,E2 28358.268} C_VEL
LIN {X 0,Y 743.916,Z 1197.735,A -85,B 0,C 180,E1 28356.173,E2 28356.173} C_VEL
LIN {X 0,Y 743.909,Z 1201.928,A -85,B 0,C 180,E1 28354.008,E2 28354.008} C_VEL
LIN {X 0,Y 743.912,Z 1204.213,A -85,B 0,C 180,E1 28352.003,E2 28352.003} C_VEL
LIN {X 0,Y 743.898,Z 1204.939,A -85,B 0,C 180,E1 28349.769,E2 28349.769} C_VEL
LIN {X 0,Y 743.908,Z 1203.979,A -85,B 0,C 180,E1 28347.689,E2 28347.689} C_VEL
LIN {X 0,Y 743.912,Z 1201.303,A -85,B 0,C 180,E1 28345.606,E2 28345.606} C_VEL
LIN {X 0,Y 743.919,Z 1197.152,A -85,B 0,C 180,E1 28343.595,E2 28343.595} C_VEL
LIN {X 0,Y 743.924,Z 1191.153,A -85,B 0,C 180,E1 28341.498,E2 28341.498} C_VEL
LIN {X 0,Y 743.919,Z 1183.317,A -85,B 0,C 180,E1 28339.389,E2 28339.389} C_VEL
LIN {X 0,Y 743.966,Z 1173.522,A -85,B 0,C 180,E1 28337.267,E2 28337.267} C_VEL
LIN {X 0,Y 743.999,Z 1164.522,A -85,B 0,C 180,E1 28335.604,E2 28335.604} C_VEL
LIN {X 0,Y 744.02,Z 1154.734,A -85,B 0,C 180,E1 28334.008,E2 28334.008} C_VEL
LIN {X 0,Y 744.097,Z 1144.248,A -85,B 0,C 180,E1 28332.482,E2 28332.482} C_VEL
LIN {X 0,Y 744.155,Z 1131.862,A -85,B 0,C 180,E1 28330.862,E2 28330.862} C_VEL
LIN {X 0,Y 744.287,Z 1114.951,A -85,B 0,C 180,E1 28328.898,E2 28328.898} C_VEL
LIN {X 0,Y 744.424,Z 1098.824,A -85,B 0,C 180,E1 28327.243,E2 28327.243} C_VEL
LIN {X 0,Y 744.541,Z 1082.149,A -85,B 0,C 180,E1 28325.691,E2 28325.691} C_VEL
LIN {X 0,Y 744.781,Z 1061.264,A -85,B 0,C 180,E1 28323.96,E2 28323.96} C_VEL
LIN {X 0,Y 744.926,Z 1043.435,A -85,B 0,C 180,E1 28322.631,E2 28322.631} C_VEL
LIN {X 0,Y 745.124,Z 1024.604,A -85,B 0,C 180,E1 28321.356,E2 28321.356} C_VEL
LIN {X 0,Y 745.416,Z 1000.231,A -85,B 0,C 180,E1 28319.889,E2 28319.889} C_VEL
LIN {X 0,Y 745.617,Z 979.491,A -85,B 0,C 180,E1 28318.786,E2 28318.786} C_VEL
LIN {X 0,Y 745.813,Z 959.68,A -85,B 0,C 180,E1 28317.843,E2 28317.843} C_VEL
LIN {X 0,Y 746.014,Z 938.347,A -85,B 0,C 180,E1 28316.941,E2 28316.941} C_VEL
LIN {X 0,Y 746.299,Z 911.417,A -85,B 0,C 180,E1 28315.965,E2 28315.965} C_VEL
LIN {X 0,Y 746.495,Z 885.148,A -85,B 0,C 180,E1 28315.178,E2 28315.178} C_VEL
LIN {X 0,Y 746.663,Z 858.693,A -85,B 0,C 180,E1 28314.547,E2 28314.547} C_VEL
LIN {X 0,Y 746.818,Z 832.214,A -85,B 0,C 180,E1 28314.07,E2 28314.07} C_VEL
LIN {X 0,Y 746.939,Z 789.963,A -85,B 0,C 180,E1 28313.549,E2 28313.549} C_VEL
LIN {X 0,Y 747.381,Z 562.694,A -85,B 0,C 180,E1 28310.868,E2 28310.868} C_VEL
LIN {X 0,Y 747.807,Z 354.264,A -85,B 0,C 180,E1 28308.319,E2 28308.319} C_VEL
LIN {X 0,Y 746.81,Z 349.256,A -85,B 0,C 180,E1 28308.146,E2 28308.146} C_VEL
LIN {X 0,Y 746.953,Z 318.638,A -85,B 0,C 180,E1 28306.291,E2 28306.291} C_VEL
LIN {X 0,Y 744.01,Z 311.985,A -85,B 0,C 180,E1 28305.641,E2 28305.641} C_VEL
LIN {X 0,Y 743.971,Z 311.489,A -85,B 0,C 180,E1 28305.232,E2 28305.232} C_VEL
LIN {X 0,Y 743.968,Z 311.555,A -85,B 0,C 180,E1 28302.222,E2 28302.222} C_VEL
LIN {X 0,Y 743.946,Z 311.55,A -85,B 0,C 180,E1 28299.755,E2 28299.755} C_VEL
LIN {X 0,Y 743.957,Z 311.555,A -85,B 0,C 180,E1 28297.409,E2 28297.409} C_VEL
LIN {X 0,Y 744.038,Z 311.551,A -85,B 0,C 180,E1 28294.549,E2 28294.549} C_VEL
LIN {X 0,Y 743.966,Z 311.549,A -85,B 0,C 180,E1 28291.793,E2 28291.793} C_VEL
LIN {X 0,Y 743.968,Z 311.553,A -85,B 0,C 180,E1 28289.289,E2 28289.289} C_VEL
LIN {X 0,Y 744.038,Z 311.552,A -85,B 0,C 180,E1 28286.491,E2 28286.491} C_VEL
LIN {X 0,Y 743.981,Z 311.544,A -85,B 0,C 180,E1 28283.694,E2 28283.694} C_VEL
LIN {X 0,Y 743.982,Z 311.551,A -85,B 0,C 180,E1 28281.112,E2 28281.112} C_VEL
LIN {X 0,Y 744.034,Z 311.546,A -85,B 0,C 180,E1 28278.329,E2 28278.329} C_VEL
LIN {X 0,Y 743.992,Z 311.547,A -85,B 0,C 180,E1 28275.506,E2 28275.506} C_VEL
LIN {X 0,Y 744.001,Z 311.551,A -85,B 0,C 180,E1 28272.812,E2 28272.812} C_VEL
LIN {X 0,Y 744.039,Z 311.543,A -85,B 0,C 180,E1 28269.827,E2 28269.827} C_VEL
LIN {X 0,Y 743.994,Z 311.547,A -85,B 0,C 180,E1 28267.025,E2 28267.025} C_VEL
LIN {X 0,Y 744.032,Z 311.553,A -85,B 0,C 180,E1 28264.239,E2 28264.239} C_VEL
LIN {X 0,Y 744.016,Z 311.543,A -85,B 0,C 180,E1 28261.309,E2 28261.309} C_VEL
LIN {X 0,Y 744.032,Z 311.55,A -85,B 0,C 180,E1 28258.383,E2 28258.383} C_VEL
LIN {X 0,Y 744.032,Z 311.541,A -85,B 0,C 180,E1 28255.298,E2 28255.298} C_VEL
LIN {X 0,Y 744.034,Z 311.549,A -85,B 0,C 180,E1 28252.277,E2 28252.277} C_VEL
LIN {X 0,Y 744.015,Z 311.548,A -85,B 0,C 180,E1 28251.802,E2 28251.802} C_VEL
LIN {X 0,Y 743.035,Z 311.669,A -85,B 0,C 180,E1 28251.209,E2 28251.209} C_VEL
LIN {X 0,Y 736.648,Z 312.463,A -85,B 0,C 180,E1 28249.547,E2 28249.547} C_VEL
LIN {X 0,Y 736.093,Z 312.53,A -85,B 0,C 180,E1 28249.116,E2 28249.116} C_VEL
LIN {X 0,Y 736.093,Z 312.54,A -85,B 0,C 180,E1 28246.088,E2 28246.088} C_VEL
LIN {X 0,Y 736.092,Z 312.53,A -85,B 0,C 180,E1 28243.1,E2 28243.1} C_VEL
LIN {X 0,Y 736.088,Z 312.544,A -85,B 0,C 180,E1 28239.982,E2 28239.982} C_VEL
LIN {X 0,Y 736.081,Z 312.53,A -85,B 0,C 180,E1 28237.054,E2 28237.054} C_VEL
LIN {X 0,Y 736.093,Z 312.545,A -85,B 0,C 180,E1 28233.975,E2 28233.975} C_VEL
LIN {X 0,Y 736.062,Z 312.529,A -85,B 0,C 180,E1 28231.079,E2 28231.079} C_VEL
LIN {X 0,Y 736.092,Z 312.541,A -85,B 0,C 180,E1 28228.193,E2 28228.193} C_VEL
LIN {X 0,Y 736.051,Z 312.542,A -85,B 0,C 180,E1 28225.401,E2 28225.401} C_VEL
LIN {X 0,Y 736.069,Z 312.53,A -85,B 0,C 180,E1 28222.709,E2 28222.709} C_VEL
LIN {X 0,Y 736.066,Z 312.536,A -85,B 0,C 180,E1 28219.611,E2 28219.611} C_VEL
LIN {X 0,Y 736.038,Z 312.542,A -85,B 0,C 180,E1 28216.958,E2 28216.958} C_VEL
LIN {X 0,Y 736.101,Z 312.538,A -85,B 0,C 180,E1 28214.173,E2 28214.173} C_VEL
LIN {X 0,Y 736.092,Z 312.778,A -85,B 0,C 180,E1 28213.474,E2 28213.474} C_VEL
LIN {X 0,Y 737.575,Z 316.364,A -85,B 0,C 180,E1 28213.097,E2 28213.097} C_VEL
LIN {X 0,Y 740.205,Z 322.819,A -85,B 0,C 180,E1 28212.486,E2 28212.486} C_VEL
LIN {X 0,Y 739.704,Z 363.194,A -85,B 0,C 180,E1 28209.946,E2 28209.946} C_VEL
LIN {X 0,Y 739.507,Z 396.954,A -85,B 0,C 180,E1 28207.904,E2 28207.904} C_VEL
LIN {X 0,Y 740.693,Z 403.032,A -85,B 0,C 180,E1 28207.756,E2 28207.756} C_VEL
LIN {X 0,Y 740.055,Z 648.45,A -85,B 0,C 180,E1 28204.896,E2 28204.896} C_VEL
LIN {X 0,Y 739.565,Z 829.567,A -85,B 0,C 180,E1 28202.823,E2 28202.823} C_VEL
LIN {X 0,Y 739.427,Z 851.829,A -85,B 0,C 180,E1 28202.465,E2 28202.465} C_VEL
LIN {X 0,Y 739.152,Z 878.679,A -85,B 0,C 180,E1 28201.876,E2 28201.876} C_VEL
LIN {X 0,Y 738.942,Z 900.026,A -85,B 0,C 180,E1 28201.281,E2 28201.281} C_VEL
LIN {X 0,Y 738.717,Z 921.007,A -85,B 0,C 180,E1 28200.587,E2 28200.587} C_VEL
LIN {X 0,Y 738.382,Z 945.912,A -85,B 0,C 180,E1 28199.614,E2 28199.614} C_VEL
LIN {X 0,Y 738.072,Z 967.668,A -85,B 0,C 180,E1 28198.613,E2 28198.613} C_VEL
LIN {X 0,Y 737.806,Z 988.527,A -85,B 0,C 180,E1 28197.524,E2 28197.524} C_VEL
LIN {X 0,Y 737.433,Z 1011.443,A -85,B 0,C 180,E1 28196.154,E2 28196.154} C_VEL
LIN {X 0,Y 737.186,Z 1029.974,A -85,B 0,C 180,E1 28194.9,E2 28194.9} C_VEL
LIN {X 0,Y 736.896,Z 1051.286,A -85,B 0,C 180,E1 28193.274,E2 28193.274} C_VEL
LIN {X 0,Y 736.693,Z 1067.564,A -85,B 0,C 180,E1 28191.874,E2 28191.874} C_VEL
LIN {X 0,Y 736.475,Z 1085.275,A -85,B 0,C 180,E1 28190.172,E2 28190.172} C_VEL
LIN {X 0,Y 736.32,Z 1100.304,A -85,B 0,C 180,E1 28188.528,E2 28188.528} C_VEL
LIN {X 0,Y 736.199,Z 1114.275,A -85,B 0,C 180,E1 28186.816,E2 28186.816} C_VEL
LIN {X 0,Y 736.081,Z 1127.421,A -85,B 0,C 180,E1 28184.957,E2 28184.957} C_VEL
LIN {X 0,Y 736.023,Z 1137.338,A -85,B 0,C 180,E1 28183.353,E2 28183.353} C_VEL
LIN {X 0,Y 735.979,Z 1146.374,A -85,B 0,C 180,E1 28181.679,E2 28181.679} C_VEL
LIN {X 0,Y 735.923,Z 1155.675,A -85,B 0,C 180,E1 28179.62,E2 28179.62} C_VEL
LIN {X 0,Y 735.928,Z 1161.99,A -85,B 0,C 180,E1 28177.887,E2 28177.887} C_VEL
LIN {X 0,Y 735.922,Z 1166.827,A -85,B 0,C 180,E1 28176.24,E2 28176.24} C_VEL
LIN {X 0,Y 735.905,Z 1171.166,A -85,B 0,C 180,E1 28174.286,E2 28174.286} C_VEL
LIN {X 0,Y 735.914,Z 1173.831,A -85,B 0,C 180,E1 28172.258,E2 28172.258} C_VEL
LIN {X 0,Y 735.891,Z 1174.814,A -85,B 0,C 180,E1 28170.623,E2 28170.623} C_VEL
LIN {X 0,Y 735.91,Z 1174.706,A -85,B 0,C 180,E1 28168.91,E2 28168.91} C_VEL
LIN {X 0,Y 735.908,Z 1172.918,A -85,B 0,C 180,E1 28166.807,E2 28166.807} C_VEL
LIN {X 0,Y 735.901,Z 1170.076,A -85,B 0,C 180,E1 28165.09,E2 28165.09} C_VEL
LIN {X 0,Y 735.915,Z 1166.239,A -85,B 0,C 180,E1 28163.447,E2 28163.447} C_VEL
LIN {X 0,Y 735.93,Z 1161.007,A -85,B 0,C 180,E1 28161.72,E2 28161.72} C_VEL
LIN {X 0,Y 735.954,Z 1152.717,A -85,B 0,C 180,E1 28159.59,E2 28159.59} C_VEL
LIN {X 0,Y 735.978,Z 1144.793,A -85,B 0,C 180,E1 28157.924,E2 28157.924} C_VEL
LIN {X 0,Y 736.017,Z 1136.005,A -85,B 0,C 180,E1 28156.327,E2 28156.327} C_VEL
LIN {X 0,Y 736.128,Z 1123.737,A -85,B 0,C 180,E1 28154.399,E2 28154.399} C_VEL
LIN {X 0,Y 736.208,Z 1111.135,A -85,B 0,C 180,E1 28152.697,E2 28152.697} C_VEL
LIN {X 0,Y 736.331,Z 1098.248,A -85,B 0,C 180,E1 28151.145,E2 28151.145} C_VEL
LIN {X 0,Y 736.546,Z 1080.746,A -85,B 0,C 180,E1 28149.285,E2 28149.285} C_VEL
LIN {X 0,Y 736.693,Z 1065.309,A -85,B 0,C 180,E1 28147.833,E2 28147.833} C_VEL
LIN {X 0,Y 736.978,Z 1046.992,A -85,B 0,C 180,E1 28146.284,E2 28146.284} C_VEL
LIN {X 0,Y 737.215,Z 1027.528,A -85,B 0,C 180,E1 28144.837,E2 28144.837} C_VEL
LIN {X 0,Y 737.536,Z 1007.141,A -85,B 0,C 180,E1 28143.48,E2 28143.48} C_VEL
LIN {X 0,Y 737.824,Z 985.369,A -85,B 0,C 180,E1 28142.214,E2 28142.214} C_VEL
LIN {X 0,Y 738.092,Z 965.04,A -85,B 0,C 180,E1 28141.167,E2 28141.167} C_VEL
LIN {X 0,Y 738.486,Z 940.24,A -85,B 0,C 180,E1 28140.06,E2 28140.06} C_VEL
LIN {X 0,Y 738.731,Z 918.303,A -85,B 0,C 180,E1 28139.228,E2 28139.228} C_VEL
LIN {X 0,Y 738.961,Z 897.009,A -85,B 0,C 180,E1 28138.537,E2 28138.537} C_VEL
LIN {X 0,Y 739.272,Z 870.835,A -85,B 0,C 180,E1 28137.843,E2 28137.843} C_VEL
LIN {X 0,Y 739.446,Z 847.797,A -85,B 0,C 180,E1 28137.374,E2 28137.374} C_VEL
LIN {X 0,Y 739.571,Z 827.506,A -85,B 0,C 180,E1 28137.06,E2 28137.06} C_VEL
LIN {X 0,Y 740.246,Z 573.031,A -85,B 0,C 180,E1 28134.146,E2 28134.146} C_VEL
LIN {X 0,Y 740.621,Z 401.785,A -85,B 0,C 180,E1 28132.135,E2 28132.135} C_VEL
LIN {X 0,Y 739.407,Z 396.015,A -85,B 0,C 180,E1 28131.966,E2 28131.966} C_VEL
LIN {X 0,Y 739.883,Z 351.141,A -85,B 0,C 180,E1 28129.217,E2 28129.217} C_VEL
LIN {X 0,Y 740.056,Z 322.065,A -85,B 0,C 180,E1 28127.365,E2 28127.365} C_VEL
LIN {X 0,Y 736.109,Z 312.918,A -85,B 0,C 180,E1 28126.458,E2 28126.458} C_VEL
LIN {X 0,Y 736.099,Z 312.531,A -85,B 0,C 180,E1 28125.935,E2 28125.935} C_VEL
LIN {X 0,Y 736.033,Z 312.542,A -85,B 0,C 180,E1 28123.104,E2 28123.104} C_VEL
LIN {X 0,Y 736.039,Z 312.534,A -85,B 0,C 180,E1 28120.591,E2 28120.591} C_VEL
LIN {X 0,Y 736.096,Z 312.532,A -85,B 0,C 180,E1 28117.762,E2 28117.762} C_VEL
LIN {X 0,Y 736.047,Z 312.539,A -85,B 0,C 180,E1 28114.979,E2 28114.979} C_VEL
LIN {X 0,Y 736.064,Z 312.537,A -85,B 0,C 180,E1 28112.267,E2 28112.267} C_VEL
LIN {X 0,Y 736.085,Z 312.527,A -85,B 0,C 180,E1 28109.187,E2 28109.187} C_VEL
LIN {X 0,Y 736.057,Z 312.541,A -85,B 0,C 180,E1 28106.373,E2 28106.373} C_VEL
LIN {X 0,Y 736.088,Z 312.535,A -85,B 0,C 180,E1 28103.524,E2 28103.524} C_VEL
LIN {X 0,Y 736.065,Z 312.536,A -85,B 0,C 180,E1 28100.683,E2 28100.683} C_VEL
LIN {X 0,Y 736.094,Z 312.536,A -85,B 0,C 180,E1 28097.786,E2 28097.786} C_VEL
LIN {X 0,Y 736.09,Z 312.532,A -85,B 0,C 180,E1 28094.796,E2 28094.796} C_VEL
LIN {X 0,Y 736.095,Z 312.535,A -85,B 0,C 180,E1 28091.757,E2 28091.757} C_VEL
LIN {X 0,Y 736.093,Z 312.531,A -85,B 0,C 180,E1 28088.672,E2 28088.672} C_VEL
LIN {X 0,Y 736.092,Z 312.537,A -85,B 0,C 180,E1 28085.613,E2 28085.613} C_VEL
LIN {X 0,Y 736.094,Z 312.531,A -85,B 0,C 180,E1 28082.569,E2 28082.569} C_VEL
LIN {X 0,Y 736.09,Z 312.537,A -85,B 0,C 180,E1 28079.533,E2 28079.533} C_VEL
LIN {X 0,Y 736.083,Z 312.533,A -85,B 0,C 180,E1 28076.573,E2 28076.573} C_VEL
LIN {X 0,Y 736.096,Z 312.535,A -85,B 0,C 180,E1 28073.526,E2 28073.526} C_VEL
LIN {X 0,Y 736.058,Z 312.536,A -85,B 0,C 180,E1 28070.697,E2 28070.697} C_VEL
LIN {X 0,Y 736.09,Z 312.532,A -85,B 0,C 180,E1 28067.845,E2 28067.845} C_VEL
LIN {X 0,Y 736.053,Z 312.541,A -85,B 0,C 180,E1 28064.981,E2 28064.981} C_VEL
LIN {X 0,Y 736.074,Z 312.528,A -85,B 0,C 180,E1 28062.203,E2 28062.203} C_VEL
LIN {X 0,Y 736.067,Z 312.542,A -85,B 0,C 180,E1 28059.151,E2 28059.151} C_VEL
LIN {X 0,Y 736.036,Z 312.533,A -85,B 0,C 180,E1 28056.485,E2 28056.485} C_VEL
LIN {X 0,Y 736.098,Z 312.537,A -85,B 0,C 180,E1 28053.703,E2 28053.703} C_VEL
LIN {X 0,Y 736.038,Z 312.542,A -85,B 0,C 180,E1 28050.811,E2 28050.811} C_VEL
LIN {X 0,Y 736.026,Z 312.538,A -85,B 0,C 180,E1 28048.282,E2 28048.282} C_VEL
LIN {X 0,Y 736.095,Z 312.539,A -85,B 0,C 180,E1 28045.497,E2 28045.497} C_VEL
LIN {X 0,Y 736.021,Z 312.544,A -85,B 0,C 180,E1 28042.609,E2 28042.609} C_VEL
LIN {X 0,Y 736.009,Z 312.538,A -85,B 0,C 180,E1 28040.218,E2 28040.218} C_VEL
LIN {X 0,Y 736.034,Z 312.545,A -85,B 0,C 180,E1 28037.743,E2 28037.743} C_VEL
LIN {X 0,Y 736.089,Z 312.681,A -85,B 0,C 180,E1 28034.95,E2 28034.95} C_VEL
LIN {X 0,Y 737.288,Z 315.939,A -85,B 0,C 180,E1 28034.603,E2 28034.603} C_VEL
LIN {X 0,Y 740.617,Z 323.166,A -85,B 0,C 180,E1 28033.895,E2 28033.895} C_VEL
LIN {X 0,Y 740.444,Z 350.706,A -85,B 0,C 180,E1 28032.238,E2 28032.238} C_VEL
LIN {X 0,Y 741.808,Z 357.151,A -85,B 0,C 180,E1 28032.058,E2 28032.058} C_VEL
LIN {X 0,Y 741.139,Z 569.897,A -85,B 0,C 180,E1 28029.438,E2 28029.438} C_VEL
LIN {X 0,Y 740.477,Z 795.344,A -85,B 0,C 180,E1 28026.757,E2 28026.757} C_VEL
LIN {X 0,Y 740.311,Z 833.628,A -85,B 0,C 180,E1 28026.274,E2 28026.274} C_VEL
LIN {X 0,Y 740.075,Z 860.29,A -85,B 0,C 180,E1 28025.782,E2 28025.782} C_VEL
LIN {X 0,Y 739.82,Z 886.262,A -85,B 0,C 180,E1 28025.152,E2 28025.152} C_VEL
LIN {X 0,Y 739.497,Z 914.343,A -85,B 0,C 180,E1 28024.295,E2 28024.295} C_VEL
LIN {X 0,Y 739.092,Z 939.477,A -85,B 0,C 180,E1 28023.362,E2 28023.362} C_VEL
LIN {X 0,Y 738.79,Z 960.685,A -85,B 0,C 180,E1 28022.454,E2 28022.454} C_VEL
LIN {X 0,Y 738.489,Z 981.245,A -85,B 0,C 180,E1 28021.46,E2 28021.46} C_VEL
LIN {X 0,Y 738.11,Z 1005.689,A -85,B 0,C 180,E1 28020.125,E2 28020.125} C_VEL
LIN {X 0,Y 737.733,Z 1026.903,A -85,B 0,C 180,E1 28018.804,E2 28018.804} C_VEL
LIN {X 0,Y 737.448,Z 1045.341,A -85,B 0,C 180,E1 28017.532,E2 28017.532} C_VEL
LIN {X 0,Y 737.181,Z 1066.232,A -85,B 0,C 180,E1 28015.937,E2 28015.937} C_VEL
LIN {X 0,Y 736.851,Z 1085.145,A -85,B 0,C 180,E1 28014.305,E2 28014.305} C_VEL
LIN {X 0,Y 736.68,Z 1100.569,A -85,B 0,C 180,E1 28012.838,E2 28012.838} C_VEL
LIN {X 0,Y 736.469,Z 1117.988,A -85,B 0,C 180,E1 28011.003,E2 28011.003} C_VEL
LIN {X 0,Y 736.295,Z 1132.512,A -85,B 0,C 180,E1 28009.268,E2 28009.268} C_VEL
LIN {X 0,Y 736.196,Z 1144.252,A -85,B 0,C 180,E1 28007.712,E2 28007.712} C_VEL
LIN {X 0,Y 736.091,Z 1154.738,A -85,B 0,C 180,E1 28006.168,E2 28006.168} C_VEL
LIN {X 0,Y 736.044,Z 1164.525,A -85,B 0,C 180,E1 28004.555,E2 28004.555} C_VEL
LIN {X 0,Y 735.988,Z 1174.755,A -85,B 0,C 180,E1 28002.634,E2 28002.634} C_VEL
LIN {X 0,Y 735.948,Z 1184.913,A -85,B 0,C 180,E1 28000.331,E2 28000.331} C_VEL
LIN {X 0,Y 735.928,Z 1192.136,A -85,B 0,C 180,E1 27998.28,E2 27998.28} C_VEL
